C07324=1177.921,389.608,-82.395,-176.029,8.968,148.653
C07325=1177.916,389.855,-82.431,-176.029,8.971,148.654
C07326=1177.913,390.103,-82.467,-176.029,8.974,148.654
C07327=1177.909,390.350,-82.502,-176.028,8.977,148.655
C07328=1177.905,390.597,-82.538,-176.028,8.979,148.656
C07329=1177.901,390.845,-82.573,-176.028,8.983,148.657
C07330=1177.897,391.093,-82.609,-176.027,8.985,148.657
C07331=1177.893,391.340,-82.645,-176.027,8.988,148.658
C07332=1177.889,391.623,-82.686,-176.027,8.991,148.659
C07333=1177.884,391.908,-82.727,-176.027,8.994,148.659
C07334=1177.880,392.193,-82.768,-176.026,8.998,148.660
C07335=1177.874,392.477,-82.808,-176.026,9.001,148.661
C07336=1177.871,392.724,-82.844,-176.026,9.004,148.662
C07337=1177.867,392.972,-82.880,-176.026,9.006,148.662
C07338=1177.863,393.219,-82.915,-176.026,9.009,148.663
C07339=1177.860,393.467,-82.951,-176.026,9.012,148.664
C07340=1177.855,393.714,-82.986,-176.025,9.014,148.664
C07341=1177.851,393.961,-83.023,-176.025,9.017,148.665
C07342=1177.848,394.208,-83.058,-176.025,9.020,148.666
C07343=1177.844,394.456,-83.094,-176.025,9.022,148.666
C07344=1177.840,394.704,-83.130,-176.025,9.025,148.667
C07345=1177.836,394.951,-83.166,-176.025,9.027,148.668
C07346=1177.832,395.198,-83.201,-176.025,9.031,148.668
C07347=1177.827,395.446,-83.237,-176.025,9.033,148.669
C07348=1177.824,395.693,-83.272,-176.025,9.036,148.670
C07349=1177.820,395.941,-83.308,-176.025,9.038,148.670
C07350=1177.816,396.188,-83.343,-176.025,9.040,148.671
C07351=1177.811,396.435,-83.379,-176.025,9.043,148.672
C07352=1177.808,396.682,-83.416,-176.025,9.046,148.672
C07353=1177.804,396.930,-83.451,-176.024,9.049,148.673
C07354=1177.800,397.178,-83.487,-176.024,9.051,148.674
C07355=1177.796,397.425,-83.523,-176.025,9.054,148.674
C07356=1177.793,397.673,-83.558,-176.024,9.056,148.675
C07357=1177.789,397.920,-83.594,-176.024,9.059,148.676
C07358=1177.784,398.167,-83.630,-176.025,9.061,148.676
C07359=1177.780,398.415,-83.665,-176.024,9.064,148.677
C07360=1177.777,398.662,-83.701,-176.024,9.066,148.677
C07361=1177.773,398.909,-83.738,-176.025,9.069,148.678
C07362=1177.769,399.157,-83.773,-176.024,9.071,148.679
C07363=1177.765,399.404,-83.809,-176.025,9.073,148.679
C07364=1177.760,399.652,-83.844,-176.025,9.076,148.680
C07365=1177.757,399.899,-83.880,-176.025,9.077,148.681
C07366=1177.753,400.146,-83.916,-176.025,9.080,148.681
C07367=1177.749,400.394,-83.952,-176.025,9.083,148.682
C07368=1177.745,400.641,-83.988,-176.025,9.085,148.683
C07369=1177.741,400.889,-84.023,-176.025,9.087,148.683
C07370=1177.737,401.137,-84.060,-176.025,9.090,148.684
C07371=1177.733,401.383,-84.096,-176.025,9.092,148.685
C07372=1177.729,401.630,-84.131,-176.025,9.095,148.685
C07373=1177.725,401.878,-84.167,-176.026,9.096,148.686
C07374=1177.721,402.126,-84.203,-176.026,9.099,148.686
C07375=1177.718,402.373,-84.238,-176.026,9.101,148.687
C07376=1177.714,402.620,-84.275,-176.026,9.104,148.688
C07377=1177.710,402.868,-84.311,-176.026,9.106,148.688
C07378=1177.706,403.115,-84.346,-176.026,9.108,148.689
C07379=1177.701,403.362,-84.382,-176.026,9.110,148.690
C07380=1177.698,403.610,-84.418,-176.026,9.113,148.690
C07381=1177.694,403.857,-84.454,-176.026,9.115,148.691
C07382=1177.690,404.105,-84.490,-176.027,9.117,148.691
C07383=1177.686,404.352,-84.526,-176.027,9.119,148.692
C07384=1177.682,404.600,-84.562,-176.027,9.122,148.693
C07385=1177.678,404.847,-84.598,-176.027,9.124,148.693
C07386=1177.675,405.094,-84.634,-176.027,9.126,148.694
C07387=1177.670,405.341,-84.669,-176.027,9.128,148.694
C07388=1177.666,405.589,-84.705,-176.027,9.131,148.695
C07389=1177.663,405.836,-84.741,-176.027,9.132,148.696
C07390=1177.658,406.084,-84.777,-176.028,9.135,148.696
C07391=1177.655,406.331,-84.813,-176.027,9.137,148.697
C07392=1177.651,406.578,-84.850,-176.028,9.139,148.697
C07393=1177.647,406.826,-84.885,-176.028,9.141,148.698
C07394=1177.643,407.073,-84.921,-176.028,9.143,148.699
C07395=1177.639,407.321,-84.957,-176.028,9.145,148.699
C07396=1177.636,407.568,-84.993,-176.028,9.147,148.700
C07397=1177.631,407.815,-85.028,-176.029,9.149,148.700
C07398=1177.627,408.063,-85.064,-176.029,9.151,148.701
C07399=1177.624,408.309,-85.101,-176.029,9.154,148.702
C07400=1177.619,408.557,-85.137,-176.029,9.155,148.702
C07401=1177.615,408.805,-85.172,-176.029,9.158,148.703
C07402=1177.612,409.052,-85.209,-176.030,9.159,148.703
C07403=1177.608,409.299,-85.245,-176.029,9.162,148.704
C07404=1177.604,409.547,-85.280,-176.030,9.163,148.704
C07405=1177.600,409.795,-85.317,-176.030,9.166,148.705
C07406=1177.596,410.042,-85.353,-176.030,9.167,148.706
C07407=1177.592,410.289,-85.389,-176.030,9.170,148.706
C07408=1177.588,410.536,-85.424,-176.030,9.172,148.707
C07409=1177.584,410.783,-85.460,-176.030,9.173,148.707
C07410=1177.580,411.031,-85.497,-176.031,9.176,148.708
C07411=1177.576,411.278,-85.532,-176.031,9.177,148.708
C07412=1177.572,411.526,-85.569,-176.031,9.180,148.709
C07413=1177.568,411.773,-85.604,-176.031,9.181,148.710
C07414=1177.565,412.021,-85.640,-176.031,9.184,148.710
C07415=1177.561,412.268,-85.677,-176.031,9.185,148.711
C07416=1177.557,412.515,-85.712,-176.031,9.188,148.711
C07417=1177.553,412.762,-85.749,-176.032,9.189,148.712
C07418=1177.549,413.010,-85.785,-176.032,9.191,148.712
C07419=1177.545,413.258,-85.821,-176.032,9.193,148.713
C07420=1177.541,413.504,-85.857,-176.033,9.194,148.713
C07421=1177.537,413.752,-85.893,-176.032,9.197,148.714
C07422=1177.533,413.999,-85.929,-176.033,9.198,148.714
C07423=1177.529,414.246,-85.965,-176.033,9.201,148.715
C07424=1177.525,414.494,-86.001,-176.033,9.202,148.715
C07425=1177.522,414.741,-86.037,-176.033,9.204,148.716
C07426=1177.517,414.989,-86.073,-176.033,9.206,148.716
C07427=1177.514,415.236,-86.109,-176.033,9.208,148.717
C07428=1177.510,415.475,-86.144,-176.033,9.210,148.718
C07429=1177.506,415.715,-86.178,-176.034,9.211,148.718
C07430=1177.503,415.955,-86.214,-176.033,9.214,148.719
C07431=1177.502,416.194,-86.248,-176.034,9.215,148.719
C07432=1177.502,416.433,-86.283,-176.034,9.216,148.720
C07433=1177.502,416.672,-86.318,-176.034,9.219,148.720
C07434=1177.505,416.911,-86.352,-176.034,9.220,148.720
C07435=1177.507,417.150,-86.386,-176.034,9.222,148.721
C07436=1177.086,417.151,-86.429,-176.037,9.232,148.725
C07437=1177.083,416.911,-86.395,-176.037,9.231,148.724
C07438=1177.081,416.670,-86.360,-176.037,9.229,148.724
C07439=1177.081,416.430,-86.326,-176.037,9.227,148.723
C07440=1177.081,416.189,-86.291,-176.037,9.226,148.723
C07441=1177.082,415.948,-86.256,-176.036,9.224,148.722
C07442=1177.085,415.707,-86.221,-176.037,9.222,148.722
C07443=1177.088,415.466,-86.186,-176.036,9.221,148.721
C07444=1177.092,415.225,-86.151,-176.036,9.219,148.721
C07445=1177.097,414.977,-86.115,-176.036,9.217,148.720
C07446=1177.100,414.730,-86.079,-176.036,9.215,148.720
C07447=1177.104,414.483,-86.042,-176.036,9.213,148.719
C07448=1177.108,414.235,-86.007,-176.036,9.211,148.719
C07449=1177.112,413.988,-85.970,-176.036,9.209,148.718
C07450=1177.116,413.741,-85.934,-176.036,9.208,148.718
C07451=1177.119,413.493,-85.899,-176.035,9.206,148.717
C07452=1177.123,413.246,-85.862,-176.035,9.204,148.716
C07453=1177.127,412.998,-85.826,-176.035,9.202,148.716
C07454=1177.132,412.751,-85.790,-176.035,9.200,148.715
C07455=1177.135,412.504,-85.754,-176.034,9.198,148.715
C07456=1177.140,412.257,-85.718,-176.035,9.196,148.714
C07457=1177.143,412.010,-85.682,-176.034,9.194,148.714
C07458=1177.148,411.762,-85.646,-176.034,9.192,148.713
C07459=1177.151,411.514,-85.610,-176.034,9.191,148.713
C07460=1177.155,411.267,-85.574,-176.034,9.188,148.712
C07461=1177.159,411.020,-85.538,-176.034,9.187,148.712
C07462=1177.163,410.772,-85.502,-176.034,9.184,148.711
C07463=1177.167,410.525,-85.465,-176.033,9.183,148.710
C07464=1177.170,410.277,-85.430,-176.033,9.180,148.710
C07465=1177.175,410.030,-85.394,-176.033,9.179,148.709
C07466=1177.178,409.783,-85.357,-176.033,9.176,148.709
C07467=1177.182,409.536,-85.322,-176.033,9.175,148.708
C07468=1177.187,409.288,-85.286,-176.032,9.172,148.708
C07469=1177.190,409.041,-85.250,-176.032,9.171,148.707
C07470=1177.195,408.793,-85.214,-176.032,9.168,148.706
C07471=1177.198,408.546,-85.178,-176.032,9.166,148.706
C07472=1177.202,408.299,-85.142,-176.032,9.164,148.705
C07473=1177.206,408.051,-85.106,-176.032,9.162,148.705
C07474=1177.210,407.804,-85.070,-176.031,9.160,148.704
C07475=1177.214,407.557,-85.033,-176.031,9.158,148.703
C07476=1177.217,407.309,-84.998,-176.032,9.156,148.703
C07477=1177.221,407.062,-84.962,-176.031,9.154,148.702
C07478=1177.226,406.815,-84.926,-176.031,9.152,148.702
C07479=1177.230,406.568,-84.890,-176.030,9.150,148.701
C07480=1177.234,406.320,-84.854,-176.031,9.148,148.701
C07481=1177.238,406.072,-84.818,-176.031,9.145,148.700
C07482=1177.241,405.825,-84.782,-176.030,9.143,148.699
C07483=1177.245,405.578,-84.746,-176.030,9.141,148.699
C07484=1177.249,405.330,-84.710,-176.030,9.139,148.698
C07485=1177.253,405.082,-84.674,-176.030,9.137,148.698
C07486=1177.257,404.835,-84.638,-176.029,9.135,148.697
C07487=1177.261,404.589,-84.603,-176.030,9.132,148.696
C07488=1177.265,404.341,-84.567,-176.029,9.131,148.696
C07489=1177.269,404.093,-84.531,-176.029,9.128,148.695
C07490=1177.272,403.846,-84.495,-176.029,9.126,148.694
C07491=1177.277,403.599,-84.459,-176.029,9.123,148.694
C07492=1177.281,403.351,-84.423,-176.029,9.122,148.693
C07493=1177.285,403.103,-84.387,-176.029,9.119,148.693
C07494=1177.288,402.856,-84.351,-176.029,9.117,148.692
C07495=1177.292,402.609,-84.315,-176.029,9.114,148.691
C07496=1177.297,402.362,-84.279,-176.028,9.113,148.691
C07497=1177.301,402.114,-84.244,-176.028,9.110,148.690
C07498=1177.304,401.867,-84.208,-176.028,9.108,148.689
C07499=1177.308,401.620,-84.172,-176.028,9.106,148.689
C07500=1177.312,401.372,-84.136,-176.028,9.103,148.688
C07501=1177.316,401.125,-84.100,-176.027,9.101,148.687
C07502=1177.320,400.877,-84.064,-176.028,9.099,148.687
C07503=1177.324,400.631,-84.028,-176.027,9.096,148.686
C07504=1177.328,400.383,-83.993,-176.027,9.094,148.686
C07505=1177.332,400.135,-83.957,-176.028,9.092,148.685
C07506=1177.336,399.888,-83.921,-176.027,9.089,148.684
C07507=1177.339,399.640,-83.886,-176.027,9.086,148.684
C07508=1177.344,399.393,-83.849,-176.028,9.084,148.683
C07509=1177.347,399.146,-83.813,-176.027,9.082,148.682
C07510=1177.351,398.898,-83.778,-176.027,9.079,148.682
C07511=1177.356,398.651,-83.742,-176.027,9.077,148.681
C07512=1177.359,398.404,-83.706,-176.027,9.074,148.680
C07513=1177.363,398.156,-83.671,-176.027,9.072,148.680
C07514=1177.367,397.909,-83.634,-176.027,9.069,148.679
C07515=1177.371,397.661,-83.598,-176.027,9.067,148.678
C07516=1177.375,397.414,-83.563,-176.027,9.064,148.678
C07517=1177.380,397.167,-83.527,-176.027,9.062,148.677
C07518=1177.383,396.919,-83.491,-176.027,9.059,148.676
C07519=1177.387,396.672,-83.456,-176.027,9.057,148.676
C07520=1177.391,396.424,-83.420,-176.027,9.054,148.675
C07521=1177.395,396.177,-83.384,-176.027,9.052,148.675
C07522=1177.398,395.930,-83.348,-176.027,9.049,148.674
C07523=1177.403,395.683,-83.313,-176.027,9.047,148.673
C07524=1177.407,395.435,-83.277,-176.027,9.045,148.673
C07525=1177.411,395.187,-83.241,-176.027,9.041,148.672
C07526=1177.414,394.940,-83.206,-176.027,9.039,148.671
C07527=1177.418,394.692,-83.170,-176.027,9.036,148.670
C07528=1177.422,394.445,-83.134,-176.027,9.034,148.670
C07529=1177.427,394.198,-83.099,-176.027,9.031,148.669
C07530=1177.430,393.950,-83.063,-176.028,9.028,148.668
C07531=1177.434,393.703,-83.027,-176.028,9.026,148.668
C07532=1177.438,393.456,-82.991,-176.028,9.023,148.667
C07533=1177.442,393.208,-82.955,-176.028,9.020,148.666
C07534=1177.445,392.961,-82.920,-176.028,9.017,148.666
C07535=1177.450,392.714,-82.884,-176.028,9.015,148.665
C07536=1177.454,392.466,-82.848,-176.028,9.012,148.664
C07537=1177.458,392.181,-82.808,-176.028,9.009,148.664
C07538=1177.463,391.897,-82.766,-176.029,9.005,148.663
C07539=1177.467,391.613,-82.726,-176.029,9.002,148.662
C07540=1177.472,391.328,-82.684,-176.029,8.999,148.661
C07541=1177.476,391.081,-82.649,-176.029,8.996,148.661
C07542=1177.479,390.833,-82.613,-176.030,8.994,148.660
C07543=1177.484,390.587,-82.578,-176.030,8.990,148.659
C07544=1177.487,390.339,-82.543,-176.030,8.988,148.659
C07545=1177.492,390.091,-82.506,-176.031,8.985,148.658
C07546=1177.495,389.844,-82.471,-176.031,8.982,148.657
C07547=1177.499,389.596,-82.435,-176.031,8.979,148.657
C07548=1177.503,389.350,-82.400,-176.031,8.977,148.656
C07549=1177.507,389.102,-82.365,-176.032,8.973,148.655
C07550=1177.511,388.854,-82.328,-176.033,8.970,148.655
C07551=1177.515,388.607,-82.293,-176.032,8.967,148.654
C07552=1177.519,388.360,-82.258,-176.033,8.964,148.653
C07553=1177.523,388.112,-82.223,-176.034,8.961,148.652
C07554=1177.527,387.864,-82.187,-176.034,8.959,148.652
C07555=1177.531,387.617,-82.152,-176.034,8.955,148.651
C07556=1177.535,387.369,-82.116,-176.035,8.952,148.651
C07557=1177.539,387.122,-82.080,-176.035,8.949,148.650
C07558=1177.543,386.875,-82.045,-176.036,8.947,148.649
C07559=1177.547,386.627,-82.009,-176.036,8.943,148.649
C07560=1177.550,386.380,-81.974,-176.037,8.940,148.648
C07561=1177.554,386.133,-81.939,-176.037,8.937,148.647
C07562=1177.558,385.885,-81.903,-176.038,8.934,148.647
C07563=1177.563,385.637,-81.868,-176.038,8.931,148.646
C07564=1177.567,385.390,-81.832,-176.039,8.928,148.645
C07565=1177.571,385.143,-81.797,-176.040,8.925,148.645
C07566=1177.574,384.895,-81.761,-176.040,8.921,148.644
C07567=1177.578,384.648,-81.726,-176.041,8.918,148.643
C07568=1177.582,384.401,-81.691,-176.042,8.915,148.643
C07569=1177.586,384.153,-81.655,-176.042,8.912,148.642
C07570=1177.590,383.905,-81.620,-176.043,8.909,148.641
C07571=1177.594,383.658,-81.585,-176.044,8.906,148.641
C07572=1177.599,383.411,-81.549,-176.044,8.902,148.640
C07573=1177.602,383.163,-81.513,-176.045,8.899,148.639
C07574=1177.606,382.915,-81.479,-176.046,8.896,148.639
C07575=1177.610,382.668,-81.443,-176.047,8.892,148.638
C07576=1177.614,382.421,-81.408,-176.048,8.889,148.637
C07577=1177.618,382.173,-81.372,-176.048,8.886,148.637
C07578=1177.622,381.926,-81.337,-176.049,8.883,148.636
C07579=1177.626,381.678,-81.302,-176.050,8.880,148.636
C07580=1177.630,381.431,-81.267,-176.051,8.876,148.635
C07581=1177.633,381.183,-81.231,-176.052,8.873,148.635
C07582=1177.638,380.936,-81.197,-176.053,8.869,148.634
C07583=1177.642,380.688,-81.161,-176.054,8.866,148.633
C07584=1177.645,380.441,-81.126,-176.054,8.863,148.633
C07585=1177.650,380.194,-81.091,-176.056,8.859,148.632
C07586=1177.654,379.946,-81.056,-176.057,8.856,148.631
C07587=1177.657,379.698,-81.020,-176.057,8.853,148.631
C07588=1177.662,379.451,-80.986,-176.059,8.849,148.630
C07589=1177.665,379.204,-80.950,-176.060,8.846,148.630
C07590=1177.669,378.956,-80.914,-176.060,8.843,148.629
C07591=1177.674,378.709,-80.880,-176.062,8.839,148.628
C07592=1177.677,378.461,-80.844,-176.063,8.836,148.628
C07593=1177.681,378.214,-80.809,-176.064,8.832,148.627
C07594=1177.686,377.966,-80.774,-176.065,8.829,148.627
C07595=1177.689,377.719,-80.739,-176.066,8.825,148.626
C07596=1177.693,377.471,-80.704,-176.068,8.822,148.626
C07597=1177.697,377.224,-80.669,-176.068,8.819,148.625
C07598=1177.701,376.976,-80.634,-176.070,8.815,148.624
C07599=1177.705,376.728,-80.598,-176.071,8.812,148.624
C07600=1177.709,376.481,-80.563,-176.072,8.808,148.623
C07601=1177.713,376.233,-80.528,-176.074,8.804,148.623
C07602=1177.718,375.986,-80.493,-176.075,8.801,148.622
C07603=1177.722,375.738,-80.458,-176.076,8.797,148.622
C07604=1177.724,375.491,-80.423,-176.077,8.794,148.621
C07605=1177.729,375.244,-80.389,-176.079,8.791,148.621
C07606=1177.733,374.996,-80.353,-176.080,8.788,148.620
C07607=1177.737,374.749,-80.319,-176.081,8.784,148.619
C07608=1177.741,374.501,-80.283,-176.083,8.780,148.619
C07609=1177.745,374.253,-80.249,-176.084,8.777,148.618
C07610=1177.749,374.006,-80.214,-176.085,8.773,148.618
C07611=1177.753,373.758,-80.179,-176.087,8.769,148.617
C07612=1177.757,373.511,-80.145,-176.088,8.766,148.617
C07613=1177.761,373.264,-80.109,-176.089,8.763,148.616
C07614=1177.765,373.016,-80.074,-176.091,8.759,148.616
C07615=1177.769,372.768,-80.040,-176.092,8.756,148.615
C07616=1177.773,372.521,-80.004,-176.094,8.752,148.615
C07617=1177.777,372.273,-79.970,-176.095,8.748,148.614
C07618=1177.780,372.026,-79.935,-176.097,8.745,148.613
C07619=1177.785,371.779,-79.900,-176.099,8.741,148.613
C07620=1177.789,371.530,-79.866,-176.099,8.738,148.612
C07621=1177.793,371.282,-79.831,-176.101,8.734,148.612
C07622=1177.797,371.036,-79.796,-176.103,8.731,148.612
C07623=1177.800,370.788,-79.761,-176.104,8.727,148.611
C07624=1177.805,370.540,-79.727,-176.106,8.723,148.611
C07625=1177.809,370.293,-79.691,-176.108,8.720,148.610
C07626=1177.813,370.045,-79.657,-176.109,8.716,148.610
C07627=1177.816,369.798,-79.623,-176.111,8.713,148.609
C07628=1177.821,369.550,-79.588,-176.113,8.709,148.609
C07629=1177.825,369.303,-79.553,-176.114,8.706,148.608
C07630=1177.829,369.055,-79.518,-176.116,8.702,148.608
C07631=1177.832,368.807,-79.484,-176.118,8.698,148.607
C07632=1177.837,368.560,-79.449,-176.119,8.695,148.607
C07633=1177.841,368.312,-79.415,-176.121,8.692,148.606
C07634=1177.844,368.065,-79.380,-176.123,8.688,148.606
C07635=1177.848,367.817,-79.345,-176.124,8.684,148.606
C07636=1177.853,367.570,-79.311,-176.126,8.681,148.605
C07637=1177.856,367.322,-79.277,-176.128,8.677,148.605
C07638=1177.861,367.075,-79.242,-176.130,8.674,148.604
C07639=1177.865,366.827,-79.207,-176.132,8.670,148.604
C07640=1177.869,366.579,-79.173,-176.134,8.666,148.603
C07641=1177.873,366.298,-79.134,-176.135,8.662,148.603
C07642=1177.878,366.016,-79.094,-176.137,8.658,148.602
C07643=1177.882,365.734,-79.055,-176.140,8.653,148.602
C07644=1177.887,365.452,-79.016,-176.142,8.650,148.601
C07645=1177.891,365.205,-78.981,-176.143,8.646,148.601
C07646=1177.895,364.957,-78.947,-176.145,8.643,148.600
C07647=1177.899,364.710,-78.913,-176.147,8.639,148.600
C07648=1177.902,364.462,-78.878,-176.149,8.636,148.600
C07649=1177.907,364.215,-78.844,-176.151,8.632,148.599
C07650=1177.911,363.968,-78.810,-176.153,8.628,148.599
C07651=1177.915,363.719,-78.775,-176.155,8.625,148.599
C07652=1177.919,363.472,-78.741,-176.157,8.622,148.598
C07653=1177.923,363.224,-78.707,-176.159,8.618,148.598
C07654=1177.927,362.976,-78.673,-176.161,8.614,148.597
C07655=1177.931,362.729,-78.639,-176.163,8.611,148.597
C07656=1177.935,362.481,-78.604,-176.165,8.607,148.597
C07657=1177.939,362.234,-78.570,-176.167,8.603,148.596
C07658=1177.943,361.986,-78.535,-176.169,8.599,148.596
C07659=1177.947,361.739,-78.501,-176.171,8.596,148.596
C07660=1177.951,361.491,-78.467,-176.173,8.592,148.595
C07661=1177.955,361.243,-78.433,-176.175,8.589,148.595
C07662=1177.960,360.995,-78.399,-176.177,8.585,148.595
C07663=1177.963,360.748,-78.365,-176.179,8.582,148.594
C07664=1177.967,360.500,-78.331,-176.181,8.579,148.594
C07665=1177.971,360.253,-78.296,-176.183,8.575,148.593
C07666=1177.975,360.005,-78.263,-176.185,8.572,148.593
C07667=1177.979,359.757,-78.228,-176.188,8.567,148.593
C07668=1177.983,359.510,-78.195,-176.190,8.564,148.593
C07669=1177.988,359.263,-78.160,-176.192,8.560,148.592
C07670=1177.991,359.014,-78.127,-176.194,8.557,148.592
C07671=1177.995,358.767,-78.093,-176.196,8.553,148.591
C07672=1178.000,358.520,-78.058,-176.198,8.550,148.591
C07673=1178.003,358.271,-78.025,-176.200,8.546,148.591
C07674=1178.008,358.024,-77.990,-176.202,8.543,148.591
C07675=1178.012,357.777,-77.956,-176.205,8.539,148.590
C07676=1178.015,357.528,-77.923,-176.207,8.535,148.590
C07677=1178.020,357.281,-77.888,-176.209,8.532,148.590
C07678=1178.024,357.033,-77.855,-176.211,8.528,148.589
C07679=1178.028,356.786,-77.821,-176.213,8.525,148.589
C07680=1178.032,356.538,-77.787,-176.216,8.522,148.589
C07681=1178.036,356.290,-77.753,-176.217,8.518,148.588
C07682=1178.040,356.043,-77.720,-176.220,8.514,148.588
C07683=1178.044,355.794,-77.685,-176.223,8.511,148.588
C07684=1178.048,355.547,-77.652,-176.224,8.507,148.587
C07685=1178.052,355.299,-77.618,-176.227,8.504,148.587
C07686=1178.056,355.052,-77.584,-176.229,8.501,148.587
C07687=1178.060,354.804,-77.550,-176.231,8.497,148.587
C07688=1178.064,354.556,-77.517,-176.233,8.494,148.586
C07689=1178.068,354.309,-77.483,-176.235,8.490,148.586
C07690=1178.072,354.062,-77.449,-176.238,8.486,148.586
C07691=1178.077,353.814,-77.416,-176.240,8.483,148.586
C07692=1178.080,353.565,-77.382,-176.242,8.479,148.585
C07693=1178.084,353.318,-77.348,-176.245,8.476,148.585
C07694=1178.088,353.070,-77.315,-176.247,8.473,148.585
C07695=1178.093,352.823,-77.281,-176.249,8.469,148.585
C07696=1178.097,352.575,-77.248,-176.251,8.466,148.584
C07697=1178.100,352.327,-77.214,-176.253,8.462,148.584
C07698=1178.104,352.080,-77.180,-176.256,8.458,148.584
C07699=1178.108,351.832,-77.147,-176.258,8.455,148.583
C07700=1178.113,351.584,-77.113,-176.261,8.452,148.583
C07701=1178.117,351.337,-77.079,-176.262,8.448,148.583
C07702=1178.121,351.089,-77.046,-176.265,8.445,148.583
C07703=1178.125,350.841,-77.013,-176.267,8.441,148.582
C07704=1178.129,350.593,-76.980,-176.269,8.438,148.582
C07705=1178.133,350.346,-76.946,-176.271,8.435,148.582
C07706=1178.137,350.098,-76.913,-176.274,8.431,148.582
C07707=1178.141,349.850,-76.879,-176.277,8.427,148.581
C07708=1178.146,349.602,-76.846,-176.279,8.424,148.581
C07709=1178.150,349.355,-76.812,-176.281,8.420,148.581
C07710=1178.153,349.107,-76.778,-176.283,8.417,148.581
C07711=1178.157,348.859,-76.745,-176.285,8.414,148.580
C07712=1178.161,348.611,-76.712,-176.287,8.410,148.580
C07713=1178.166,348.364,-76.679,-176.290,8.407,148.580
C07714=1178.170,348.116,-76.646,-176.292,8.404,148.580
C07715=1178.174,347.868,-76.612,-176.294,8.401,148.579
C07716=1178.178,347.620,-76.579,-176.296,8.397,148.579
C07717=1178.182,347.373,-76.545,-176.299,8.393,148.579
C07718=1178.186,347.125,-76.512,-176.302,8.390,148.579
C07719=1178.190,346.878,-76.479,-176.304,8.386,148.579
C07720=1178.194,346.630,-76.446,-176.306,8.383,148.578
C07721=1178.198,346.382,-76.413,-176.308,8.380,148.578
C07722=1178.202,346.134,-76.379,-176.311,8.377,148.578
C07723=1178.206,345.886,-76.346,-176.313,8.373,148.578
C07724=1178.210,345.638,-76.313,-176.315,8.370,148.577
C07725=1178.214,345.391,-76.280,-176.317,8.367,148.577
C07726=1178.219,345.143,-76.247,-176.320,8.363,148.577
C07727=1178.223,344.895,-76.214,-176.322,8.360,148.577
C07728=1178.227,344.647,-76.180,-176.324,8.357,148.577
C07729=1178.231,344.399,-76.148,-176.327,8.353,148.576
C07730=1178.235,344.151,-76.115,-176.329,8.349,148.576
C07731=1178.240,343.904,-76.082,-176.332,8.346,148.576
C07732=1178.244,343.656,-76.048,-176.334,8.343,148.576
C07733=1178.248,343.408,-76.015,-176.336,8.339,148.576
C07734=1178.252,343.160,-75.982,-176.338,8.336,148.575
C07735=1178.255,342.913,-75.950,-176.341,8.333,148.575
C07736=1178.259,342.665,-75.916,-176.343,8.329,148.575
C07737=1178.264,342.417,-75.884,-176.345,8.326,148.575
C07738=1178.268,342.169,-75.851,-176.348,8.323,148.575
C07739=1178.272,341.922,-75.818,-176.350,8.320,148.574
C07740=1178.276,341.674,-75.785,-176.353,8.316,148.574
C07741=1178.281,341.425,-75.752,-176.355,8.313,148.574
C07742=1178.284,341.178,-75.719,-176.357,8.310,148.574
C07743=1178.289,340.931,-75.687,-176.359,8.307,148.574
C07744=1178.293,340.683,-75.654,-176.362,8.302,148.573
C07745=1178.298,340.404,-75.616,-176.364,8.299,148.573
C07746=1178.302,340.125,-75.580,-176.368,8.295,148.573
C07747=1178.307,339.845,-75.543,-176.370,8.292,148.573
C07748=1178.311,339.566,-75.506,-176.373,8.288,148.573
C07749=1178.316,339.319,-75.473,-176.375,8.285,148.572
C07750=1178.320,339.070,-75.440,-176.377,8.281,148.572
C07751=1178.323,338.823,-75.408,-176.380,8.278,148.572
C07752=1178.328,338.575,-75.375,-176.382,8.275,148.572
C07753=1178.332,338.327,-75.342,-176.385,8.272,148.572
C07754=1178.336,338.079,-75.309,-176.387,8.268,148.572
C07755=1178.340,337.832,-75.278,-176.389,8.265,148.571
C07756=1178.345,337.584,-75.245,-176.391,8.262,148.571
C07757=1178.349,337.336,-75.212,-176.394,8.259,148.571
C07758=1178.352,337.088,-75.180,-176.396,8.255,148.571
C07759=1178.357,336.841,-75.146,-176.399,8.252,148.571
C07760=1178.361,336.592,-75.114,-176.401,8.249,148.570
C07761=1178.364,336.345,-75.081,-176.404,8.246,148.570
C07762=1178.369,336.096,-75.049,-176.406,8.242,148.570
C07763=1178.374,335.849,-75.016,-176.409,8.238,148.570
C07764=1178.377,335.601,-74.984,-176.411,8.235,148.570
C07765=1178.382,335.353,-74.952,-176.414,8.232,148.570
C07766=1178.385,335.106,-74.919,-176.416,8.229,148.570
C07767=1178.390,334.857,-74.887,-176.418,8.225,148.569
C07768=1178.394,334.609,-74.854,-176.421,8.222,148.569
C07769=1178.398,334.362,-74.822,-176.423,8.219,148.569
C07770=1178.403,334.114,-74.790,-176.426,8.216,148.569
C07771=1178.406,333.866,-74.757,-176.428,8.212,148.569
C07772=1178.410,333.618,-74.725,-176.430,8.209,148.569
C07773=1178.414,333.370,-74.693,-176.433,8.206,148.569
C07774=1178.419,333.123,-74.660,-176.435,8.203,148.568
C07775=1178.423,332.875,-74.628,-176.437,8.200,148.568
C07776=1178.427,332.627,-74.596,-176.440,8.197,148.568
C07777=1178.431,332.379,-74.563,-176.442,8.193,148.568
C07778=1178.435,332.131,-74.531,-176.445,8.190,148.568
C07779=1178.440,331.883,-74.499,-176.447,8.187,148.568
C07780=1178.444,331.635,-74.467,-176.450,8.184,148.567
C07781=1178.448,331.387,-74.434,-176.452,8.180,148.567
C07782=1178.451,331.139,-74.402,-176.455,8.177,148.567
C07783=1178.456,330.892,-74.370,-176.457,8.174,148.567
C07784=1178.460,330.644,-74.338,-176.459,8.171,148.567
C07785=1178.465,330.395,-74.306,-176.462,8.168,148.567
C07786=1178.468,330.148,-74.273,-176.464,8.164,148.567
C07787=1178.472,329.901,-74.242,-176.466,8.161,148.566
C07788=1178.477,329.652,-74.209,-176.469,8.158,148.566
C07789=1178.480,329.404,-74.177,-176.471,8.155,148.566
C07790=1178.485,329.156,-74.145,-176.474,8.152,148.566
C07791=1178.489,328.908,-74.113,-176.476,8.148,148.566
C07792=1178.493,328.660,-74.081,-176.479,8.145,148.566
C07793=1178.497,328.412,-74.049,-176.481,8.142,148.566
C07794=1178.502,328.165,-74.018,-176.484,8.139,148.566
C07795=1178.506,327.916,-73.985,-176.486,8.136,148.566
C07796=1178.510,327.668,-73.953,-176.489,8.133,148.565
C07797=1178.514,327.421,-73.922,-176.491,8.129,148.565
C07798=1178.519,327.173,-73.889,-176.494,8.126,148.565
C07799=1178.522,326.925,-73.858,-176.496,8.123,148.565
C07800=1178.527,326.677,-73.826,-176.498,8.120,148.565
C07801=1178.531,326.429,-73.794,-176.501,8.117,148.565
C07802=1178.535,326.181,-73.762,-176.503,8.114,148.565
C07803=1178.539,325.934,-73.730,-176.506,8.110,148.565
C07804=1178.543,325.685,-73.698,-176.508,8.107,148.564
C07805=1178.547,325.437,-73.666,-176.511,8.104,148.564
C07806=1178.551,325.190,-73.635,-176.513,8.101,148.564
C07807=1178.555,324.942,-73.603,-176.516,8.098,148.564
C07808=1178.560,324.693,-73.570,-176.518,8.094,148.564
C07809=1178.564,324.446,-73.539,-176.521,8.091,148.564
C07810=1178.568,324.197,-73.508,-176.523,8.088,148.564
C07811=1178.572,323.949,-73.476,-176.526,8.085,148.564
C07812=1178.577,323.702,-73.444,-176.528,8.082,148.564
C07813=1178.580,323.454,-73.412,-176.531,8.079,148.564
C07814=1178.585,323.206,-73.380,-176.533,8.075,148.563
C07815=1178.588,322.958,-73.349,-176.536,8.072,148.563
C07816=1178.592,322.710,-73.317,-176.538,8.069,148.563
C07817=1178.597,322.462,-73.285,-176.541,8.066,148.563
C07818=1178.601,322.214,-73.253,-176.543,8.063,148.563
C07819=1178.605,321.967,-73.222,-176.546,8.060,148.563
C07820=1178.610,321.718,-73.191,-176.548,8.057,148.563
C07821=1178.614,321.471,-73.159,-176.551,8.054,148.563
C07822=1178.618,321.223,-73.128,-176.553,8.050,148.563
C07823=1178.622,320.974,-73.096,-176.556,8.047,148.563
C07824=1178.627,320.726,-73.064,-176.558,8.044,148.562
C07825=1178.630,320.478,-73.032,-176.561,8.041,148.562
C07826=1178.635,320.230,-73.002,-176.563,8.038,148.562
C07827=1178.639,319.982,-72.970,-176.566,8.035,148.562
C07828=1178.643,319.734,-72.939,-176.568,8.031,148.562
C07829=1178.647,319.486,-72.907,-176.571,8.028,148.562
C07830=1178.651,319.239,-72.876,-176.573,8.025,148.562
C07831=1178.655,318.990,-72.845,-176.576,8.022,148.562
C07832=1178.660,318.743,-72.813,-176.578,8.019,148.562
C07833=1178.664,318.494,-72.782,-176.581,8.016,148.562
C07834=1178.668,318.247,-72.751,-176.583,8.012,148.561
C07835=1178.672,317.998,-72.719,-176.586,8.009,148.562
C07836=1178.676,317.751,-72.688,-176.588,8.007,148.562
C07837=1178.680,317.502,-72.657,-176.590,8.004,148.561
C07838=1178.685,317.255,-72.625,-176.593,8.001,148.561
C07839=1178.689,317.006,-72.594,-176.595,7.998,148.561
C07840=1178.693,316.759,-72.563,-176.598,7.995,148.561
C07841=1178.697,316.510,-72.532,-176.600,7.991,148.561
C07842=1178.701,316.263,-72.500,-176.603,7.988,148.561
C07843=1178.705,316.014,-72.469,-176.605,7.985,148.561
C07844=1178.710,315.766,-72.438,-176.608,7.982,148.561
C07845=1178.714,315.519,-72.407,-176.610,7.979,148.561
C07846=1178.718,315.270,-72.376,-176.613,7.976,148.561
C07847=1178.723,315.022,-72.345,-176.615,7.973,148.561
C07848=1178.726,314.774,-72.313,-176.618,7.970,148.561
C07849=1178.731,314.498,-72.278,-176.620,7.966,148.560
C07850=1178.736,314.220,-72.244,-176.624,7.963,148.560
C07851=1178.741,313.945,-72.210,-176.626,7.960,148.560
C07852=1178.746,313.668,-72.174,-176.629,7.956,148.560
C07853=1178.750,313.419,-72.143,-176.631,7.953,148.560
C07854=1178.754,313.171,-72.112,-176.634,7.950,148.560
C07855=1178.758,312.924,-72.082,-176.636,7.947,148.560
C07856=1178.762,312.676,-72.050,-176.639,7.944,148.560
C07857=1178.766,312.428,-72.020,-176.642,7.941,148.560
C07858=1178.770,312.179,-71.989,-176.644,7.938,148.560
C07859=1178.775,311.931,-71.958,-176.647,7.935,148.560
C07860=1178.780,311.683,-71.927,-176.649,7.931,148.560
C07861=1178.783,311.435,-71.895,-176.652,7.928,148.560
C07862=1178.787,311.187,-71.865,-176.655,7.925,148.560
C07863=1178.792,310.939,-71.834,-176.657,7.922,148.560
C07864=1178.796,310.691,-71.803,-176.659,7.919,148.560
C07865=1178.800,310.443,-71.772,-176.662,7.916,148.560
C07866=1178.804,310.195,-71.742,-176.664,7.913,148.559
C07867=1178.808,309.946,-71.711,-176.667,7.910,148.559
C07868=1178.813,309.698,-71.680,-176.669,7.908,148.559
C07869=1178.818,309.451,-71.650,-176.672,7.904,148.559
C07870=1178.821,309.202,-71.619,-176.674,7.901,148.559
C07871=1178.825,308.954,-71.588,-176.677,7.898,148.559
C07872=1178.830,308.706,-71.557,-176.679,7.895,148.559
C07873=1178.835,308.458,-71.527,-176.682,7.892,148.559
C07874=1178.838,308.210,-71.496,-176.685,7.889,148.559
C07875=1178.843,307.962,-71.465,-176.688,7.886,148.559
C07876=1178.847,307.714,-71.435,-176.690,7.883,148.559
C07877=1178.850,307.466,-71.404,-176.693,7.880,148.559
C07878=1178.855,307.218,-71.373,-176.695,7.877,148.559
C07879=1178.860,306.970,-71.343,-176.697,7.874,148.559
C07880=1178.863,306.722,-71.312,-176.700,7.871,148.559
C07881=1178.868,306.473,-71.281,-176.702,7.868,148.559
C07882=1178.872,306.225,-71.250,-176.705,7.865,148.559
C07883=1178.876,305.978,-71.220,-176.707,7.862,148.559
C07884=1178.881,305.730,-71.190,-176.710,7.859,148.559
C07885=1178.885,305.481,-71.159,-176.713,7.856,148.559
C07886=1178.889,305.233,-71.129,-176.715,7.853,148.559
C07887=1178.893,304.985,-71.098,-176.718,7.850,148.559
C07888=1178.897,304.737,-71.068,-176.721,7.847,148.559
C07889=1178.902,304.489,-71.037,-176.723,7.844,148.558
C07890=1178.906,304.240,-71.007,-176.726,7.841,148.558
C07891=1178.910,303.992,-70.977,-176.728,7.838,148.559
C07892=1178.915,303.745,-70.946,-176.730,7.835,148.559
C07893=1178.919,303.497,-70.916,-176.733,7.832,148.558
C07894=1178.924,303.248,-70.886,-176.735,7.829,148.558
C07895=1178.927,303.000,-70.855,-176.738,7.826,148.558
C07896=1178.931,302.752,-70.824,-176.741,7.823,148.558
C07897=1178.935,302.504,-70.794,-176.743,7.820,148.558
C07898=1178.940,302.256,-70.764,-176.746,7.817,148.558
C07899=1178.945,302.008,-70.733,-176.749,7.814,148.558
C07900=1178.949,301.760,-70.704,-176.751,7.812,148.558
C07901=1178.953,301.512,-70.674,-176.753,7.808,148.558
C07902=1178.957,301.263,-70.643,-176.756,7.805,148.558
C07903=1178.961,301.015,-70.613,-176.758,7.802,148.558
C07904=1178.966,300.767,-70.582,-176.761,7.799,148.558
C07905=1178.970,300.519,-70.552,-176.764,7.796,148.558
C07906=1178.974,300.271,-70.522,-176.766,7.793,148.558
C07907=1178.978,300.023,-70.492,-176.769,7.790,148.558
C07908=1178.983,299.775,-70.462,-176.772,7.787,148.558
C07909=1178.987,299.526,-70.431,-176.774,7.785,148.558
C07910=1178.991,299.278,-70.402,-176.776,7.782,148.558
C07911=1178.995,299.030,-70.371,-176.779,7.779,148.558
C07912=1179.000,298.782,-70.342,-176.782,7.776,148.558
C07913=1179.004,298.534,-70.311,-176.784,7.773,148.558
C07914=1179.008,298.285,-70.282,-176.787,7.770,148.558
C07915=1179.012,298.038,-70.251,-176.789,7.766,148.558
C07916=1179.017,297.789,-70.221,-176.792,7.763,148.558
C07917=1179.021,297.541,-70.192,-176.794,7.761,148.558
C07918=1179.025,297.293,-70.162,-176.797,7.758,148.558
C07919=1179.030,297.045,-70.132,-176.800,7.755,148.558
C07920=1179.034,296.797,-70.102,-176.802,7.752,148.558
C07921=1179.038,296.549,-70.072,-176.805,7.749,148.558
C07922=1179.042,296.300,-70.042,-176.807,7.746,148.558
C07923=1179.046,296.052,-70.012,-176.810,7.743,148.558
C07924=1179.051,295.804,-69.982,-176.812,7.741,148.558
C07925=1179.055,295.555,-69.953,-176.815,7.738,148.558
C07926=1179.059,295.307,-69.922,-176.817,7.735,148.558
C07927=1179.063,295.059,-69.892,-176.820,7.732,148.558
C07928=1179.068,294.811,-69.863,-176.823,7.729,148.558
C07929=1179.072,294.563,-69.833,-176.825,7.726,148.558
C07930=1179.076,294.315,-69.803,-176.828,7.723,148.558
C07931=1179.081,294.066,-69.773,-176.830,7.720,148.558
C07932=1179.085,293.818,-69.744,-176.833,7.717,148.558
C07933=1179.089,293.570,-69.714,-176.835,7.714,148.558
C07934=1179.093,293.322,-69.684,-176.838,7.711,148.558
C07935=1179.098,293.074,-69.654,-176.841,7.708,148.558
C07936=1179.102,292.825,-69.625,-176.843,7.705,148.558
C07937=1179.106,292.577,-69.595,-176.846,7.703,148.558
C07938=1179.110,292.329,-69.566,-176.848,7.700,148.558
C07939=1179.114,292.081,-69.536,-176.851,7.697,148.558
C07940=1179.118,291.833,-69.506,-176.853,7.694,148.558
C07941=1179.123,291.584,-69.476,-176.856,7.691,148.558
C07942=1179.128,291.337,-69.447,-176.859,7.688,148.558
C07943=1179.132,291.089,-69.418,-176.861,7.686,148.558
C07944=1179.136,290.840,-69.388,-176.864,7.683,148.558
C07945=1179.141,290.592,-69.359,-176.866,7.680,148.558
C07946=1179.145,290.344,-69.329,-176.869,7.677,148.558
C07947=1179.149,290.095,-69.300,-176.871,7.673,148.558
C07948=1179.153,289.847,-69.270,-176.874,7.670,148.558
C07949=1179.157,289.599,-69.241,-176.876,7.668,148.558
C07950=1179.162,289.351,-69.211,-176.879,7.665,148.558
C07951=1179.166,289.102,-69.182,-176.882,7.662,148.558
C07952=1179.171,288.854,-69.152,-176.884,7.659,148.558
C07953=1179.175,288.580,-69.120,-176.887,7.656,148.558
C07954=1179.180,288.305,-69.087,-176.890,7.653,148.558
C07955=1179.185,288.031,-69.055,-176.893,7.649,148.558
C07956=1179.190,287.756,-69.022,-176.896,7.646,148.558
C07957=1179.194,287.507,-68.993,-176.899,7.643,148.558
C07958=1179.198,287.259,-68.963,-176.901,7.641,148.558
C07959=1179.202,287.011,-68.934,-176.904,7.638,148.558
C07960=1179.207,286.763,-68.905,-176.906,7.635,148.558
C07961=1179.211,286.514,-68.876,-176.909,7.632,148.558
C07962=1179.216,286.266,-68.846,-176.911,7.629,148.558
C07963=1179.220,286.018,-68.817,-176.913,7.627,148.558
C07964=1179.224,285.769,-68.787,-176.916,7.624,148.558
C07965=1179.228,285.521,-68.758,-176.919,7.621,148.558
C07966=1179.233,285.273,-68.730,-176.922,7.618,148.558
C07967=1179.237,285.025,-68.700,-176.924,7.615,148.558
C07968=1179.241,284.777,-68.671,-176.927,7.613,148.559
C07969=1179.245,284.529,-68.642,-176.929,7.610,148.559
C07970=1179.249,284.280,-68.613,-176.932,7.607,148.559
C07971=1179.254,284.032,-68.584,-176.935,7.604,148.559
C07972=1179.258,283.784,-68.555,-176.937,7.601,148.559
C07973=1179.263,283.535,-68.526,-176.940,7.599,148.559
C07974=1179.267,283.287,-68.496,-176.942,7.596,148.559
C07975=1179.271,283.038,-68.467,-176.945,7.593,148.559
C07976=1179.276,282.791,-68.439,-176.947,7.589,148.559
C07977=1179.280,282.542,-68.410,-176.950,7.586,148.559
C07978=1179.284,282.294,-68.380,-176.952,7.584,148.559
C07979=1179.288,282.045,-68.351,-176.955,7.581,148.559
C07980=1179.293,281.798,-68.322,-176.958,7.578,148.559
C07981=1179.298,281.549,-68.294,-176.960,7.575,148.559
C07982=1179.301,281.301,-68.265,-176.963,7.573,148.559
C07983=1179.305,281.052,-68.235,-176.965,7.570,148.559
C07984=1179.310,280.804,-68.207,-176.968,7.567,148.559
C07985=1179.315,280.556,-68.178,-176.971,7.564,148.559
C07986=1179.319,280.307,-68.149,-176.974,7.561,148.559
C07987=1179.323,280.060,-68.120,-176.976,7.559,148.559
C07988=1179.328,279.811,-68.092,-176.978,7.556,148.559
C07989=1179.332,279.563,-68.062,-176.981,7.553,148.559
C07990=1179.336,279.314,-68.034,-176.984,7.550,148.559
C07991=1179.340,279.067,-68.005,-176.986,7.548,148.559
C07992=1179.345,278.818,-67.976,-176.989,7.545,148.559
C07993=1179.349,278.569,-67.947,-176.992,7.542,148.559
C07994=1179.353,278.322,-67.919,-176.994,7.539,148.559
C07995=1179.358,278.073,-67.890,-176.996,7.537,148.560
C07996=1179.362,277.824,-67.861,-176.999,7.534,148.560
C07997=1179.366,277.576,-67.833,-177.002,7.531,148.560
C07998=1179.371,277.328,-67.803,-177.005,7.528,148.560
C07999=1179.375,277.079,-67.775,-177.007,7.526,148.560
C08000=1179.379,276.831,-67.747,-177.009,7.523,148.560
C08001=1179.384,276.583,-67.718,-177.012,7.520,148.560
C08002=1179.387,276.335,-67.689,-177.015,7.517,148.560
C08003=1179.392,276.086,-67.661,-177.017,7.515,148.560
C08004=1179.397,275.838,-67.632,-177.020,7.512,148.560
C08005=1179.400,275.590,-67.603,-177.023,7.509,148.560
C08006=1179.405,275.341,-67.575,-177.025,7.506,148.560
C08007=1179.409,275.093,-67.547,-177.027,7.504,148.560
C08008=1179.414,274.845,-67.518,-177.030,7.501,148.560
C08009=1179.418,274.596,-67.489,-177.033,7.498,148.560
C08010=1179.422,274.348,-67.461,-177.036,7.495,148.560
C08011=1179.427,274.100,-67.433,-177.038,7.492,148.560
C08012=1179.431,273.851,-67.404,-177.041,7.489,148.560
C08013=1179.436,273.603,-67.375,-177.043,7.486,148.560
C08014=1179.440,273.355,-67.347,-177.047,7.484,148.561
C08015=1179.444,273.106,-67.318,-177.049,7.482,148.561
C08016=1179.448,272.858,-67.291,-177.051,7.479,148.561
C08017=1179.453,272.609,-67.262,-177.054,7.476,148.561
C08018=1179.457,272.361,-67.234,-177.056,7.474,148.561
C08019=1179.462,272.112,-67.205,-177.059,7.471,148.561
C08020=1179.466,271.865,-67.178,-177.062,7.468,148.561
C08021=1179.470,271.616,-67.148,-177.065,7.465,148.561
C08022=1179.475,271.368,-67.120,-177.067,7.462,148.561
C08023=1179.479,271.120,-67.092,-177.069,7.459,148.561
C08024=1179.484,270.872,-67.064,-177.072,7.457,148.561
C08025=1179.488,270.623,-67.035,-177.074,7.454,148.561
C08026=1179.492,270.375,-67.007,-177.077,7.451,148.561
C08027=1179.496,270.126,-66.979,-177.080,7.448,148.561
C08028=1179.501,269.878,-66.951,-177.083,7.445,148.562
C08029=1179.505,269.630,-66.923,-177.085,7.444,148.562
C08030=1179.510,269.381,-66.894,-177.088,7.441,148.562
C08031=1179.514,269.133,-66.866,-177.091,7.438,148.562
C08032=1179.518,268.885,-66.838,-177.093,7.435,148.562
C08033=1179.523,268.635,-66.810,-177.096,7.432,148.562
C08034=1179.527,268.388,-66.783,-177.098,7.430,148.562
C08035=1179.532,268.139,-66.754,-177.101,7.427,148.562
C08036=1179.536,267.891,-66.726,-177.103,7.424,148.562
C08037=1179.540,267.642,-66.698,-177.106,7.421,148.562
C08038=1179.545,267.394,-66.670,-177.109,7.418,148.562
C08039=1179.549,267.145,-66.641,-177.111,7.416,148.562
C08040=1179.553,266.898,-66.614,-177.114,7.414,148.563
C08041=1179.558,266.648,-66.586,-177.117,7.411,148.563
C08042=1179.562,266.400,-66.558,-177.119,7.408,148.563
C08043=1179.567,266.152,-66.530,-177.122,7.406,148.563
C08044=1179.570,265.904,-66.502,-177.124,7.403,148.563
C08045=1179.575,265.656,-66.474,-177.127,7.400,148.563
C08046=1179.579,265.406,-66.446,-177.129,7.397,148.563
C08047=1179.584,265.158,-66.418,-177.132,7.394,148.563
C08048=1179.589,264.910,-66.390,-177.135,7.393,148.563
C08049=1179.593,264.661,-66.363,-177.137,7.390,148.563
C08050=1179.597,264.413,-66.335,-177.140,7.387,148.563
C08051=1179.601,264.165,-66.307,-177.142,7.384,148.564
C08052=1179.605,263.917,-66.279,-177.145,7.381,148.564
C08053=1179.611,263.668,-66.251,-177.148,7.379,148.564
C08054=1179.615,263.419,-66.223,-177.150,7.376,148.564
C08055=1179.619,263.172,-66.195,-177.153,7.374,148.564
C08056=1179.623,262.922,-66.168,-177.156,7.371,148.564
C08057=1179.628,262.650,-66.138,-177.159,7.368,148.564
C08058=1179.633,262.376,-66.107,-177.161,7.365,148.564
C08059=1179.638,262.104,-66.077,-177.165,7.362,148.564
C08060=1179.643,261.830,-66.046,-177.167,7.359,148.565
C08061=1179.647,261.583,-66.018,-177.169,7.357,148.565
C08062=1179.651,261.333,-65.991,-177.172,7.354,148.565
C08063=1179.656,261.085,-65.963,-177.175,7.351,148.565
C08064=1179.660,260.837,-65.936,-177.177,7.349,148.565
C08065=1179.664,260.588,-65.908,-177.180,7.346,148.565
C08066=1179.669,260.340,-65.881,-177.183,7.343,148.565
C08067=1179.673,260.092,-65.853,-177.185,7.341,148.565
C08068=1179.678,259.843,-65.825,-177.188,7.338,148.565
C08069=1179.682,259.595,-65.797,-177.191,7.335,148.565
C08070=1179.687,259.346,-65.770,-177.193,7.333,148.566
C08071=1179.691,259.098,-65.742,-177.196,7.330,148.566
C08072=1179.695,258.849,-65.715,-177.199,7.327,148.566
C08073=1179.700,258.601,-65.687,-177.201,7.325,148.566
C08074=1179.704,258.353,-65.660,-177.204,7.322,148.566
C08075=1179.709,258.104,-65.633,-177.206,7.320,148.566
C08076=1179.713,257.856,-65.605,-177.209,7.317,148.566
C08077=1179.717,257.607,-65.578,-177.212,7.314,148.566
C08078=1179.722,257.359,-65.551,-177.214,7.312,148.566
C08079=1179.726,257.111,-65.523,-177.217,7.309,148.566
C08080=1179.730,256.862,-65.495,-177.220,7.307,148.567
C08081=1179.735,256.613,-65.468,-177.222,7.305,148.567
C08082=1179.739,256.365,-65.441,-177.225,7.302,148.567
C08083=1179.744,256.117,-65.414,-177.227,7.299,148.567
C08084=1179.748,255.867,-65.386,-177.230,7.296,148.567
C08085=1179.752,255.620,-65.358,-177.233,7.294,148.567
C08086=1179.757,255.371,-65.331,-177.235,7.292,148.567
C08087=1179.762,255.123,-65.304,-177.238,7.289,148.567
C08088=1179.766,254.874,-65.278,-177.240,7.287,148.568
C08089=1179.770,254.625,-65.250,-177.243,7.284,148.568
C08090=1179.774,254.377,-65.223,-177.246,7.281,148.568
C08091=1179.779,254.129,-65.195,-177.248,7.279,148.568
C08092=1179.783,253.880,-65.168,-177.251,7.276,148.568
C08093=1179.788,253.632,-65.141,-177.254,7.274,148.568
C08094=1179.792,253.383,-65.114,-177.256,7.271,148.568
C08095=1179.797,253.134,-65.087,-177.259,7.268,148.568
C08096=1179.800,252.887,-65.060,-177.261,7.266,148.569
C08097=1179.805,252.638,-65.033,-177.264,7.263,148.569
C08098=1179.810,252.390,-65.006,-177.267,7.261,148.569
C08099=1179.814,252.141,-64.979,-177.269,7.258,148.569
C08100=1179.818,251.892,-64.951,-177.272,7.255,148.569
C08101=1179.823,251.643,-64.924,-177.275,7.253,148.569
C08102=1179.827,251.395,-64.898,-177.277,7.250,148.569
C08103=1179.832,251.147,-64.870,-177.280,7.248,148.569
C08104=1179.836,250.898,-64.843,-177.283,7.246,148.570
C08105=1179.841,250.650,-64.816,-177.285,7.243,148.570
C08106=1179.846,250.401,-64.789,-177.288,7.240,148.570
C08107=1179.849,250.153,-64.763,-177.290,7.237,148.570
C08108=1179.854,249.905,-64.736,-177.293,7.236,148.570
C08109=1179.858,249.655,-64.708,-177.296,7.233,148.570
C08110=1179.863,249.407,-64.681,-177.298,7.230,148.570
C08111=1179.867,249.159,-64.655,-177.301,7.228,148.571
C08112=1179.871,248.910,-64.628,-177.303,7.226,148.571
C08113=1179.876,248.662,-64.601,-177.306,7.223,148.571
C08114=1179.880,248.414,-64.574,-177.309,7.220,148.571
C08115=1179.885,248.165,-64.547,-177.312,7.218,148.571
C08116=1179.890,247.916,-64.521,-177.314,7.215,148.571
C08117=1179.894,247.668,-64.494,-177.316,7.213,148.571
C08118=1179.898,247.419,-64.467,-177.320,7.210,148.572
C08119=1179.903,247.171,-64.440,-177.322,7.208,148.572
C08120=1179.907,246.923,-64.414,-177.325,7.205,148.572
C08121=1179.911,246.674,-64.387,-177.327,7.203,148.572
C08122=1179.916,246.425,-64.360,-177.330,7.200,148.572
C08123=1179.920,246.177,-64.334,-177.333,7.197,148.572
C08124=1179.925,245.928,-64.307,-177.335,7.195,148.573
C08125=1179.930,245.680,-64.280,-177.338,7.193,148.573
C08126=1179.934,245.432,-64.253,-177.340,7.190,148.573
C08127=1179.938,245.182,-64.227,-177.343,7.188,148.573
C08128=1179.942,244.934,-64.201,-177.346,7.186,148.573
C08129=1179.947,244.686,-64.173,-177.348,7.183,148.573
C08130=1179.952,244.437,-64.147,-177.351,7.181,148.574
C08131=1179.956,244.189,-64.121,-177.354,7.178,148.574
C08132=1179.961,243.940,-64.094,-177.356,7.176,148.574
C08133=1179.965,243.691,-64.068,-177.359,7.173,148.574
C08134=1179.969,243.443,-64.041,-177.361,7.171,148.574
C08135=1179.973,243.195,-64.014,-177.364,7.168,148.574
C08136=1179.978,242.945,-63.988,-177.367,7.166,148.574
C08137=1179.982,242.697,-63.961,-177.369,7.163,148.575
C08138=1179.987,242.449,-63.934,-177.373,7.160,148.575
C08139=1179.991,242.200,-63.909,-177.375,7.158,148.575
C08140=1179.996,241.951,-63.882,-177.378,7.155,148.575
C08141=1180.000,241.703,-63.856,-177.380,7.154,148.575
C08142=1180.005,241.454,-63.829,-177.383,7.151,148.575
C08143=1180.009,241.205,-63.803,-177.385,7.148,148.575
C08144=1180.014,240.957,-63.776,-177.388,7.146,148.576
C08145=1180.018,240.708,-63.750,-177.391,7.144,148.576
C08146=1180.022,240.460,-63.723,-177.394,7.141,148.576
C08147=1180.027,240.211,-63.697,-177.396,7.139,148.576
C08148=1180.031,239.962,-63.670,-177.399,7.136,148.576
C08149=1180.036,239.714,-63.645,-177.401,7.134,148.577
C08150=1180.040,239.466,-63.619,-177.404,7.131,148.577
C08151=1180.045,239.217,-63.592,-177.407,7.129,148.577
C08152=1180.049,238.969,-63.566,-177.409,7.126,148.577
C08153=1180.054,238.720,-63.539,-177.412,7.124,148.577
C08154=1180.058,238.471,-63.513,-177.415,7.122,148.578
C08155=1180.062,238.223,-63.487,-177.417,7.119,148.578
C08156=1180.067,237.973,-63.461,-177.420,7.117,148.578
C08157=1180.072,237.726,-63.435,-177.422,7.115,148.578
C08158=1180.076,237.477,-63.409,-177.425,7.112,148.578
C08159=1180.081,237.228,-63.383,-177.428,7.110,148.578
C08160=1180.085,236.980,-63.356,-177.430,7.108,148.578
C08161=1180.089,236.708,-63.328,-177.433,7.105,148.579
C08162=1180.094,236.436,-63.299,-177.436,7.102,148.579
C08163=1180.100,236.165,-63.271,-177.439,7.099,148.579
C08164=1180.104,235.894,-63.242,-177.442,7.097,148.579
C08165=1180.109,235.645,-63.216,-177.445,7.095,148.580
C08166=1180.113,235.396,-63.190,-177.447,7.092,148.580
C08167=1180.118,235.147,-63.164,-177.450,7.090,148.580
C08168=1180.121,234.899,-63.138,-177.453,7.087,148.580
C08169=1180.127,234.651,-63.112,-177.455,7.085,148.580
C08170=1180.131,234.402,-63.086,-177.458,7.083,148.580
C08171=1180.135,234.153,-63.061,-177.461,7.080,148.581
C08172=1180.139,233.905,-63.034,-177.463,7.078,148.581
C08173=1180.145,233.656,-63.008,-177.466,7.076,148.581
C08174=1180.149,233.408,-62.982,-177.468,7.073,148.581
C08175=1180.153,233.159,-62.957,-177.472,7.071,148.582
C08176=1180.158,232.910,-62.931,-177.474,7.069,148.582
C08177=1180.162,232.661,-62.905,-177.476,7.066,148.582
C08178=1180.167,232.413,-62.879,-177.479,7.064,148.582
C08179=1180.172,232.164,-62.853,-177.481,7.062,148.582
C08180=1180.176,231.916,-62.827,-177.485,7.059,148.582
C08181=1180.180,231.668,-62.801,-177.487,7.057,148.583
C08182=1180.185,231.419,-62.776,-177.490,7.054,148.583
C08183=1180.189,231.170,-62.750,-177.492,7.052,148.583
C08184=1180.194,230.921,-62.724,-177.495,7.050,148.583
C08185=1180.199,230.673,-62.698,-177.497,7.047,148.583
C08186=1180.203,230.424,-62.672,-177.501,7.045,148.584
C08187=1180.207,230.175,-62.647,-177.503,7.043,148.584
C08188=1180.211,229.926,-62.621,-177.506,7.041,148.584
C08189=1180.216,229.678,-62.596,-177.508,7.038,148.584
C08190=1180.220,229.429,-62.570,-177.511,7.036,148.584
C08191=1180.225,229.181,-62.544,-177.514,7.033,148.585
C08192=1180.229,228.933,-62.519,-177.516,7.031,148.585
C08193=1180.234,228.684,-62.493,-177.519,7.028,148.585
C08194=1180.238,228.434,-62.468,-177.522,7.026,148.585
C08195=1180.243,228.186,-62.443,-177.524,7.024,148.585
C08196=1180.248,227.937,-62.416,-177.527,7.022,148.586
C08197=1180.252,227.688,-62.390,-177.529,7.020,148.586
C08198=1180.257,227.440,-62.365,-177.533,7.017,148.586
C08199=1180.261,227.191,-62.339,-177.535,7.015,148.586
C08200=1180.265,226.943,-62.314,-177.537,7.013,148.587
C08201=1180.270,226.694,-62.288,-177.541,7.010,148.587
C08202=1180.275,226.445,-62.263,-177.543,7.008,148.587
C08203=1180.280,226.197,-62.238,-177.546,7.006,148.587
C08204=1180.284,225.948,-62.212,-177.548,7.003,148.587
C08205=1180.288,225.699,-62.186,-177.551,7.002,148.588
C08206=1180.292,225.452,-62.161,-177.554,6.999,148.588
C08207=1180.297,225.202,-62.136,-177.556,6.997,148.588
C08208=1180.301,224.953,-62.111,-177.559,6.994,148.588
C08209=1180.306,224.705,-62.085,-177.562,6.992,148.588
C08210=1180.310,224.456,-62.060,-177.564,6.990,148.589
C08211=1180.315,224.208,-62.035,-177.567,6.987,148.589
C08212=1180.319,223.959,-62.009,-177.570,6.986,148.589
C08213=1180.324,223.710,-61.983,-177.572,6.983,148.589
C08214=1180.329,223.461,-61.959,-177.575,6.981,148.590
C08215=1180.333,223.213,-61.933,-177.577,6.979,148.590
C08216=1180.338,222.964,-61.908,-177.580,6.976,148.590
C08217=1180.342,222.715,-61.883,-177.583,6.974,148.590
C08218=1180.346,222.467,-61.858,-177.585,6.972,148.590
C08219=1180.351,222.218,-61.833,-177.589,6.969,148.591
C08220=1180.356,221.970,-61.807,-177.591,6.967,148.591
C08221=1180.360,221.721,-61.782,-177.594,6.965,148.591
C08222=1180.364,221.471,-61.757,-177.596,6.962,148.591
C08223=1180.369,221.223,-61.731,-177.599,6.961,148.592
C08224=1180.373,220.974,-61.707,-177.602,6.958,148.592
C08225=1180.378,220.726,-61.681,-177.604,6.956,148.592
C08226=1180.382,220.477,-61.656,-177.607,6.954,148.592
C08227=1180.387,220.229,-61.631,-177.610,6.951,148.592
C08228=1180.392,219.979,-61.606,-177.612,6.949,148.593
C08229=1180.396,219.731,-61.581,-177.614,6.947,148.593
C08230=1180.400,219.482,-61.556,-177.618,6.945,148.593
C08231=1180.405,219.234,-61.531,-177.620,6.943,148.594
C08232=1180.410,218.984,-61.506,-177.623,6.940,148.594
C08233=1180.414,218.737,-61.481,-177.626,6.938,148.594
C08234=1180.418,218.487,-61.456,-177.628,6.936,148.594
C08235=1180.423,218.239,-61.430,-177.631,6.933,148.594
C08236=1180.428,217.990,-61.405,-177.634,6.931,148.595
C08237=1180.432,217.742,-61.381,-177.636,6.929,148.595
C08238=1180.436,217.492,-61.356,-177.639,6.927,148.595
C08239=1180.442,217.244,-61.331,-177.642,6.925,148.596
C08240=1180.446,216.996,-61.306,-177.644,6.923,148.596
C08241=1180.450,216.747,-61.281,-177.647,6.920,148.596
C08242=1180.455,216.498,-61.256,-177.649,6.918,148.596
C08243=1180.459,216.249,-61.231,-177.652,6.916,148.596
C08244=1180.464,216.001,-61.207,-177.655,6.914,148.597
C08245=1180.468,215.751,-61.182,-177.658,6.911,148.597
C08246=1180.473,215.503,-61.157,-177.660,6.910,148.597
C08247=1180.478,215.255,-61.132,-177.663,6.907,148.597
C08248=1180.482,215.005,-61.107,-177.666,6.905,148.598
C08249=1180.487,214.757,-61.083,-177.668,6.903,148.598
C08250=1180.491,214.508,-61.057,-177.671,6.900,148.598
C08251=1180.495,214.260,-61.033,-177.674,6.898,148.598
C08252=1180.500,214.011,-61.008,-177.676,6.897,148.599
C08253=1180.505,213.761,-60.983,-177.679,6.894,148.599
C08254=1180.509,213.514,-60.959,-177.682,6.892,148.599
C08255=1180.513,213.264,-60.934,-177.684,6.890,148.599
C08256=1180.518,213.016,-60.910,-177.687,6.887,148.600
C08257=1180.523,212.767,-60.885,-177.690,6.885,148.600
C08258=1180.527,212.518,-60.860,-177.692,6.883,148.600
C08259=1180.532,212.269,-60.836,-177.695,6.881,148.600
C08260=1180.536,212.021,-60.812,-177.698,6.879,148.601
C08261=1180.541,211.772,-60.786,-177.701,6.877,148.601
C08262=1180.546,211.523,-60.761,-177.703,6.875,148.601
C08263=1180.550,211.275,-60.737,-177.706,6.872,148.601
C08264=1180.555,211.025,-60.712,-177.709,6.870,148.602
C08265=1180.559,210.756,-60.686,-177.712,6.868,148.602
C08266=1180.564,210.485,-60.659,-177.714,6.866,148.602
C08267=1180.569,210.214,-60.633,-177.717,6.863,148.602
C08268=1180.574,209.944,-60.606,-177.720,6.861,148.603
C08269=1180.579,209.695,-60.582,-177.723,6.858,148.603
C08270=1180.583,209.446,-60.557,-177.725,6.856,148.603
C08271=1180.588,209.197,-60.532,-177.728,6.855,148.604
C08272=1180.593,208.949,-60.508,-177.731,6.853,148.604
C08273=1180.597,208.700,-60.484,-177.733,6.850,148.604
C08274=1180.602,208.451,-60.459,-177.736,6.848,148.604
C08275=1180.606,208.203,-60.435,-177.739,6.846,148.605
C08276=1180.611,207.954,-60.411,-177.742,6.844,148.605
C08277=1180.615,207.705,-60.386,-177.744,6.841,148.605
C08278=1180.619,207.456,-60.362,-177.747,6.840,148.605
C08279=1180.624,207.208,-60.337,-177.749,6.838,148.606
C08280=1180.629,206.959,-60.313,-177.752,6.835,148.606
C08281=1180.634,206.710,-60.289,-177.755,6.833,148.606
C08282=1180.638,206.461,-60.265,-177.758,6.831,148.607
C08283=1180.642,206.212,-60.241,-177.760,6.828,148.607
C08284=1180.648,205.964,-60.216,-177.763,6.827,148.607
C08285=1180.652,205.715,-60.192,-177.766,6.825,148.607
C08286=1180.656,205.466,-60.168,-177.768,6.823,148.608
C08287=1180.661,205.217,-60.144,-177.771,6.820,148.608
C08288=1180.666,204.968,-60.120,-177.774,6.818,148.608
C08289=1180.670,204.720,-60.096,-177.776,6.816,148.608
C08290=1180.675,204.471,-60.071,-177.779,6.814,148.609
C08291=1180.679,204.222,-60.046,-177.782,6.812,148.609
C08292=1180.684,203.973,-60.023,-177.784,6.810,148.609
C08293=1180.688,203.725,-59.999,-177.787,6.808,148.610
C08294=1180.693,203.476,-59.974,-177.789,6.806,148.610
C08295=1180.697,203.227,-59.950,-177.793,6.803,148.610
C08296=1180.702,202.978,-59.927,-177.795,6.802,148.610
C08297=1180.706,202.729,-59.902,-177.798,6.800,148.611
C08298=1180.711,202.481,-59.878,-177.800,6.798,148.611
C08299=1180.716,202.232,-59.854,-177.803,6.795,148.611
C08300=1180.720,201.983,-59.830,-177.806,6.793,148.612
C08301=1180.725,201.735,-59.806,-177.808,6.791,148.612
C08302=1180.729,201.485,-59.783,-177.811,6.789,148.612
C08303=1180.734,201.236,-59.758,-177.813,6.787,148.612
C08304=1180.739,200.987,-59.735,-177.817,6.785,148.613
C08305=1180.743,200.739,-59.710,-177.819,6.783,148.613
C08306=1180.747,200.490,-59.686,-177.822,6.781,148.613
C08307=1180.752,200.241,-59.663,-177.824,6.779,148.613
C08308=1180.756,199.993,-59.639,-177.827,6.777,148.614
C08309=1180.762,199.744,-59.615,-177.830,6.774,148.614
C08310=1180.766,199.495,-59.591,-177.832,6.773,148.614
C08311=1180.770,199.245,-59.567,-177.835,6.771,148.615
C08312=1180.775,198.997,-59.543,-177.838,6.769,148.615
C08313=1180.779,198.748,-59.520,-177.841,6.766,148.615
C08314=1180.784,198.500,-59.496,-177.843,6.764,148.615
C08315=1180.789,198.251,-59.472,-177.846,6.762,148.616
C08316=1180.793,198.002,-59.448,-177.848,6.761,148.616
C08317=1180.798,197.753,-59.424,-177.852,6.758,148.616
C08318=1180.803,197.504,-59.400,-177.854,6.756,148.617
C08319=1180.807,197.255,-59.377,-177.857,6.754,148.617
C08320=1180.812,197.007,-59.353,-177.859,6.752,148.617
C08321=1180.817,196.758,-59.329,-177.862,6.751,148.618
C08322=1180.821,196.509,-59.306,-177.865,6.748,148.618
C08323=1180.826,196.261,-59.282,-177.867,6.746,148.618
C08324=1180.830,196.011,-59.259,-177.870,6.744,148.618
C08325=1180.834,195.762,-59.235,-177.873,6.742,148.619
C08326=1180.839,195.513,-59.211,-177.875,6.740,148.619
C08327=1180.844,195.264,-59.187,-177.878,6.738,148.619
C08328=1180.848,195.016,-59.163,-177.881,6.736,148.620
C08329=1180.853,194.767,-59.140,-177.883,6.734,148.620
C08330=1180.857,194.518,-59.117,-177.886,6.732,148.620
C08331=1180.862,194.269,-59.093,-177.889,6.730,148.621
C08332=1180.866,194.020,-59.069,-177.891,6.728,148.621
C08333=1180.871,193.771,-59.046,-177.894,6.726,148.621
C08334=1180.876,193.522,-59.023,-177.897,6.724,148.621
C08335=1180.881,193.273,-58.999,-177.899,6.722,148.622
C08336=1180.885,193.025,-58.975,-177.902,6.720,148.622
C08337=1180.890,192.776,-58.952,-177.904,6.718,148.622
C08338=1180.895,192.528,-58.929,-177.907,6.716,148.623
C08339=1180.900,192.278,-58.905,-177.910,6.714,148.623
C08340=1180.903,192.030,-58.882,-177.913,6.712,148.623
C08341=1180.908,191.781,-58.859,-177.916,6.710,148.624
C08342=1180.913,191.532,-58.835,-177.918,6.708,148.624
C08343=1180.917,191.283,-58.812,-177.920,6.706,148.624
C08344=1180.922,191.034,-58.788,-177.923,6.704,148.624
C08345=1180.927,190.785,-58.765,-177.926,6.702,148.625
C08346=1180.931,190.536,-58.742,-177.929,6.700,148.625
C08347=1180.936,190.288,-58.718,-177.932,6.698,148.625
C08348=1180.940,190.039,-58.695,-177.934,6.696,148.626
C08349=1180.945,189.790,-58.672,-177.937,6.694,148.626
C08350=1180.949,189.541,-58.648,-177.939,6.693,148.626
C08351=1180.954,189.292,-58.625,-177.942,6.690,148.627
C08352=1180.959,189.043,-58.601,-177.945,6.688,148.627
C08353=1180.964,188.795,-58.578,-177.948,6.686,148.627
C08354=1180.968,188.546,-58.556,-177.950,6.684,148.627
C08355=1180.973,188.297,-58.532,-177.953,6.682,148.628
C08356=1180.977,188.048,-58.509,-177.955,6.681,148.628
C08357=1180.982,187.799,-58.486,-177.958,6.679,148.629
C08358=1180.987,187.550,-58.462,-177.961,6.676,148.629
C08359=1180.991,187.301,-58.440,-177.964,6.675,148.629
C08360=1180.995,187.052,-58.416,-177.967,6.673,148.630
C08361=1181.001,186.804,-58.393,-177.969,6.671,148.630
C08362=1181.005,186.555,-58.370,-177.971,6.669,148.630
C08363=1181.009,186.306,-58.347,-177.974,6.667,148.630
C08364=1181.014,186.057,-58.324,-177.977,6.665,148.631
C08365=1181.019,185.808,-58.300,-177.979,6.663,148.631
C08366=1181.023,185.558,-58.278,-177.983,6.661,148.631
C08367=1181.028,185.310,-58.255,-177.985,6.659,148.632
C08368=1181.033,185.061,-58.232,-177.988,6.657,148.632
C08369=1181.038,184.792,-58.207,-177.990,6.655,148.632
C08370=1181.043,184.522,-58.182,-177.993,6.653,148.633
C08371=1181.048,184.253,-58.157,-177.996,6.651,148.633
C08372=1181.052,183.983,-58.132,-177.999,6.649,148.634
C08373=1181.057,183.734,-58.110,-178.002,6.647,148.634
C08374=1181.062,183.485,-58.086,-178.005,6.645,148.634
C08375=1181.066,183.236,-58.063,-178.007,6.643,148.634
C08376=1181.071,182.987,-58.040,-178.010,6.641,148.635
C08377=1181.076,182.739,-58.017,-178.013,6.639,148.635
C08378=1181.080,182.489,-57.995,-178.015,6.637,148.636
C08379=1181.085,182.240,-57.972,-178.018,6.636,148.636
C08380=1181.089,181.991,-57.949,-178.021,6.634,148.636
C08381=1181.094,181.743,-57.926,-178.023,6.632,148.636
C08382=1181.099,181.493,-57.903,-178.026,6.630,148.637
C08383=1181.103,181.245,-57.881,-178.028,6.628,148.637
C08384=1181.108,180.996,-57.857,-178.031,6.626,148.637
C08385=1181.113,180.747,-57.836,-178.034,6.624,148.638
C08386=1181.118,180.498,-57.812,-178.037,6.622,148.638
C08387=1181.122,180.249,-57.789,-178.040,6.620,148.638
C08388=1181.127,180.000,-57.767,-178.042,6.619,148.639
C08389=1181.131,179.752,-57.744,-178.045,6.617,148.639
C08390=1181.136,179.503,-57.721,-178.048,6.615,148.640
C08391=1181.140,179.253,-57.699,-178.050,6.613,148.640
C08392=1181.145,179.004,-57.676,-178.052,6.611,148.640
C08393=1181.150,178.756,-57.654,-178.055,6.609,148.640
C08394=1181.154,178.507,-57.631,-178.058,6.607,148.641
C08395=1181.159,178.257,-57.608,-178.061,6.606,148.641
C08396=1181.164,178.009,-57.586,-178.063,6.604,148.642
C08397=1181.168,177.760,-57.563,-178.066,6.601,148.642
C08398=1181.173,177.511,-57.540,-178.069,6.600,148.642
C08399=1181.177,177.263,-57.518,-178.072,6.598,148.643
C08400=1181.182,177.013,-57.495,-178.074,6.596,148.643
C08401=1181.186,176.764,-57.472,-178.077,6.594,148.643
C08402=1181.192,176.515,-57.450,-178.080,6.592,148.644
C08403=1181.196,176.266,-57.427,-178.082,6.590,148.644
C08404=1181.200,176.017,-57.405,-178.085,6.589,148.644
C08405=1181.206,175.768,-57.383,-178.087,6.587,148.645
C08406=1181.210,175.519,-57.360,-178.090,6.585,148.645
C08407=1181.215,175.270,-57.338,-178.093,6.583,148.645
C08408=1181.219,175.022,-57.315,-178.095,6.581,148.646
C08409=1181.224,174.772,-57.293,-178.098,6.580,148.646
C08410=1181.228,174.523,-57.270,-178.101,6.578,148.646
C08411=1181.233,174.275,-57.248,-178.103,6.576,148.647
C08412=1181.238,174.025,-57.225,-178.106,6.574,148.647
C08413=1181.243,173.777,-57.203,-178.109,6.573,148.647
C08414=1181.247,173.528,-57.181,-178.111,6.571,148.648
C08415=1181.252,173.278,-57.158,-178.114,6.569,148.648
C08416=1181.257,173.030,-57.136,-178.117,6.567,148.649
C08417=1181.261,172.781,-57.114,-178.120,6.565,148.649
C08418=1181.267,172.532,-57.092,-178.123,6.563,148.649
C08419=1181.271,172.283,-57.069,-178.125,6.561,148.650
C08420=1181.275,172.034,-57.047,-178.128,6.559,148.650
C08421=1181.280,171.785,-57.025,-178.131,6.558,148.650
C08422=1181.285,171.535,-57.002,-178.133,6.555,148.650
C08423=1181.289,171.287,-56.980,-178.136,6.554,148.651
C08424=1181.293,171.038,-56.958,-178.138,6.552,148.651
C08425=1181.299,170.789,-56.936,-178.141,6.550,148.652
C08426=1181.303,170.540,-56.914,-178.144,6.548,148.652
C08427=1181.308,170.292,-56.891,-178.146,6.547,148.652
C08428=1181.312,170.042,-56.869,-178.149,6.545,148.653
C08429=1181.318,169.793,-56.847,-178.152,6.543,148.653
C08430=1181.322,169.544,-56.825,-178.154,6.541,148.653
C08431=1181.326,169.295,-56.803,-178.157,6.539,148.654
C08432=1181.331,169.046,-56.781,-178.160,6.538,148.654
C08433=1181.335,168.797,-56.758,-178.162,6.536,148.654
C08434=1181.341,168.548,-56.736,-178.165,6.534,148.655
C08435=1181.345,168.299,-56.714,-178.168,6.532,148.655
C08436=1181.350,168.050,-56.692,-178.170,6.531,148.656
C08437=1181.354,167.801,-56.670,-178.173,6.529,148.656
C08438=1181.359,167.553,-56.649,-178.176,6.527,148.656
C08439=1181.364,167.303,-56.626,-178.179,6.525,148.657
C08440=1181.369,167.054,-56.604,-178.181,6.523,148.657
C08441=1181.374,166.806,-56.583,-178.184,6.522,148.657
C08442=1181.378,166.556,-56.561,-178.187,6.520,148.658
C08443=1181.383,166.308,-56.539,-178.189,6.518,148.658
C08444=1181.387,166.058,-56.517,-178.192,6.516,148.659
C08445=1181.392,165.810,-56.495,-178.195,6.515,148.659
C08446=1181.396,165.560,-56.473,-178.197,6.513,148.659
C08447=1181.402,165.311,-56.451,-178.200,6.511,148.660
C08448=1181.406,165.062,-56.429,-178.203,6.509,148.660
C08449=1181.411,164.813,-56.407,-178.205,6.508,148.660
C08450=1181.415,164.564,-56.385,-178.208,6.506,148.661
C08451=1181.420,164.315,-56.363,-178.211,6.504,148.661
C08452=1181.425,164.067,-56.342,-178.213,6.502,148.661
C08453=1181.429,163.817,-56.320,-178.216,6.500,148.662
C08454=1181.434,163.569,-56.298,-178.219,6.499,148.662
C08455=1181.438,163.319,-56.276,-178.221,6.498,148.663
C08456=1181.443,163.071,-56.254,-178.224,6.496,148.663
C08457=1181.448,162.821,-56.232,-178.226,6.494,148.663
C08458=1181.453,162.572,-56.211,-178.229,6.492,148.664
C08459=1181.458,162.324,-56.190,-178.232,6.491,148.664
C08460=1181.462,162.074,-56.168,-178.234,6.489,148.664
C08461=1181.467,161.826,-56.146,-178.237,6.487,148.665
C08462=1181.471,161.576,-56.124,-178.240,6.485,148.665
C08463=1181.476,161.328,-56.102,-178.242,6.484,148.666
C08464=1181.481,161.078,-56.081,-178.245,6.482,148.666
C08465=1181.485,160.829,-56.059,-178.248,6.480,148.667
C08466=1181.490,160.580,-56.037,-178.251,6.479,148.667
C08467=1181.495,160.332,-56.016,-178.254,6.477,148.667
C08468=1181.500,160.082,-55.994,-178.256,6.475,148.668
C08469=1181.505,159.833,-55.973,-178.259,6.473,148.668
C08470=1181.509,159.584,-55.951,-178.262,6.472,148.668
C08471=1181.514,159.335,-55.929,-178.264,6.470,148.669
C08472=1181.518,159.086,-55.909,-178.267,6.468,148.669
C08473=1181.523,158.817,-55.885,-178.270,6.466,148.670
C08474=1181.528,158.548,-55.862,-178.272,6.464,148.670
C08475=1181.534,158.279,-55.838,-178.276,6.463,148.671
C08476=1181.538,158.011,-55.815,-178.278,6.461,148.671
C08477=1181.543,157.761,-55.794,-178.281,6.460,148.671
C08478=1181.548,157.513,-55.772,-178.284,6.458,148.672
C08479=1181.553,157.263,-55.751,-178.286,6.456,148.672
C08480=1181.557,157.014,-55.729,-178.289,6.454,148.672
C08481=1181.562,156.765,-55.708,-178.292,6.452,148.673
C08482=1181.567,156.515,-55.686,-178.294,6.451,148.673
C08483=1181.571,156.267,-55.665,-178.297,6.449,148.673
C08484=1181.576,156.018,-55.644,-178.300,6.447,148.674
C08485=1181.581,155.769,-55.623,-178.302,6.445,148.674
C08486=1181.585,155.520,-55.600,-178.305,6.444,148.675
C08487=1181.591,155.271,-55.579,-178.307,6.443,148.675
C08488=1181.595,155.022,-55.558,-178.310,6.441,148.676
C08489=1181.600,154.773,-55.537,-178.313,6.440,148.676
C08490=1181.604,154.524,-55.515,-178.316,6.438,148.676
C08491=1181.609,154.274,-55.494,-178.318,6.436,148.677
C08492=1181.614,154.026,-55.473,-178.321,6.434,148.677
C08493=1181.619,153.777,-55.452,-178.324,6.432,148.677
C08494=1181.623,153.528,-55.430,-178.326,6.431,148.678
C08495=1181.628,153.278,-55.409,-178.329,6.429,148.678
C08496=1181.633,153.029,-55.388,-178.332,6.427,148.679
C08497=1181.637,152.781,-55.367,-178.334,6.426,148.679
C08498=1181.643,152.531,-55.346,-178.337,6.424,148.679
C08499=1181.647,152.282,-55.324,-178.340,6.423,148.680
C08500=1181.652,152.033,-55.303,-178.342,6.421,148.680
C08501=1181.656,151.784,-55.282,-178.345,6.420,148.681
C08502=1181.661,151.535,-55.261,-178.348,6.418,148.681
C08503=1181.666,151.286,-55.240,-178.351,6.416,148.682
C08504=1181.670,151.037,-55.219,-178.353,6.414,148.682
C08505=1181.675,150.788,-55.198,-178.356,6.412,148.682
C08506=1181.680,150.538,-55.177,-178.358,6.412,148.683
C08507=1181.684,150.290,-55.156,-178.361,6.410,148.683
C08508=1181.690,150.041,-55.135,-178.363,6.408,148.683
C08509=1181.695,149.792,-55.114,-178.367,6.407,148.684
C08510=1181.698,149.543,-55.092,-178.369,6.405,148.684
C08511=1181.704,149.293,-55.071,-178.372,6.403,148.685
C08512=1181.708,149.044,-55.051,-178.375,6.401,148.685
C08513=1181.713,148.795,-55.030,-178.377,6.400,148.686
C08514=1181.718,148.546,-55.008,-178.379,6.399,148.686
C08515=1181.722,148.297,-54.988,-178.382,6.397,148.686
C08516=1181.728,148.048,-54.967,-178.385,6.395,148.687
C08517=1181.731,147.799,-54.946,-178.388,6.394,148.687
C08518=1181.736,147.550,-54.925,-178.391,6.392,148.688
C08519=1181.741,147.301,-54.904,-178.393,6.390,148.688
C08520=1181.746,147.052,-54.883,-178.396,6.388,148.688
C08521=1181.751,146.802,-54.862,-178.398,6.387,148.689
C08522=1181.756,146.553,-54.842,-178.401,6.386,148.689
C08523=1181.761,146.304,-54.821,-178.404,6.384,148.690
C08524=1181.765,146.056,-54.800,-178.406,6.382,148.690
C08525=1181.770,145.807,-54.779,-178.409,6.381,148.691
C08526=1181.774,145.558,-54.759,-178.412,6.379,148.691
C08527=1181.780,145.308,-54.738,-178.415,6.377,148.691
C08528=1181.783,145.059,-54.717,-178.417,6.376,148.692
C08529=1181.789,144.810,-54.696,-178.420,6.375,148.692
C08530=1181.793,144.561,-54.676,-178.422,6.373,148.693
C08531=1181.798,144.311,-54.655,-178.425,6.371,148.693
C08532=1181.803,144.062,-54.634,-178.428,6.370,148.694
C08533=1181.808,143.813,-54.613,-178.431,6.368,148.694
C08534=1181.812,143.565,-54.592,-178.433,6.367,148.694
C08535=1181.817,143.316,-54.571,-178.436,6.365,148.695
C08536=1181.822,143.067,-54.551,-178.438,6.363,148.695
C08537=1181.827,142.817,-54.530,-178.441,6.362,148.695
C08538=1181.831,142.568,-54.510,-178.444,6.360,148.696
C08539=1181.836,142.319,-54.489,-178.447,6.358,148.696
C08540=1181.841,142.070,-54.468,-178.449,6.358,148.697
C08541=1181.845,141.821,-54.448,-178.452,6.356,148.697
C08542=1181.851,141.571,-54.428,-178.454,6.354,148.698
C08543=1181.855,141.322,-54.407,-178.457,6.352,148.698
C08544=1181.860,141.073,-54.387,-178.460,6.351,148.699
C08545=1181.865,140.824,-54.366,-178.462,6.350,148.699
C08546=1181.869,140.575,-54.345,-178.465,6.348,148.699
C08547=1181.874,140.326,-54.325,-178.468,6.346,148.700
C08548=1181.879,140.077,-54.304,-178.470,6.345,148.700
C08549=1181.883,139.828,-54.284,-178.473,6.343,148.701
C08550=1181.888,139.579,-54.263,-178.476,6.342,148.701
C08551=1181.893,139.330,-54.242,-178.478,6.341,148.702
C08552=1181.898,139.080,-54.223,-178.481,6.339,148.702
C08553=1181.902,138.831,-54.202,-178.484,6.337,148.702
C08554=1181.907,138.582,-54.181,-178.487,6.335,148.703
C08555=1181.912,138.333,-54.161,-178.489,6.334,148.703
C08556=1181.916,138.084,-54.141,-178.492,6.333,148.704
C08557=1181.921,137.835,-54.120,-178.495,6.331,148.704
C08558=1181.926,137.585,-54.100,-178.497,6.329,148.704
C08559=1181.930,137.336,-54.080,-178.500,6.328,148.705
C08560=1181.936,137.087,-54.059,-178.502,6.327,148.705
C08561=1181.941,136.839,-54.039,-178.505,6.325,148.706
C08562=1181.945,136.589,-54.019,-178.508,6.324,148.706
C08563=1181.950,136.340,-53.999,-178.511,6.322,148.707
C08564=1181.955,136.091,-53.978,-178.513,6.320,148.707
C08565=1181.959,135.842,-53.957,-178.515,6.319,148.707
C08566=1181.964,135.593,-53.938,-178.519,6.318,148.708
C08567=1181.969,135.344,-53.917,-178.521,6.316,148.708
C08568=1181.973,135.095,-53.897,-178.524,6.314,148.709
C08569=1181.979,134.845,-53.877,-178.526,6.313,148.709
C08570=1181.983,134.596,-53.856,-178.529,6.312,148.710
C08571=1181.988,134.348,-53.836,-178.532,6.310,148.710
C08572=1181.993,134.098,-53.817,-178.535,6.308,148.711
C08573=1181.997,133.849,-53.796,-178.537,6.307,148.711
C08574=1182.003,133.599,-53.776,-178.540,6.306,148.711
C08575=1182.007,133.350,-53.756,-178.543,6.304,148.712
C08576=1182.012,133.101,-53.735,-178.545,6.303,148.712
C08577=1182.016,132.833,-53.714,-178.548,6.301,148.713
C08578=1182.022,132.564,-53.693,-178.551,6.299,148.713
C08579=1182.027,132.296,-53.671,-178.554,6.298,148.714
C08580=1182.032,132.027,-53.649,-178.557,6.296,148.714
C08581=1182.037,131.778,-53.629,-178.559,6.295,148.715
C08582=1182.042,131.529,-53.609,-178.562,6.294,148.715
C08583=1182.047,131.280,-53.589,-178.565,6.292,148.716
C08584=1182.051,131.030,-53.569,-178.567,6.290,148.716
C08585=1182.056,130.781,-53.549,-178.569,6.289,148.716
C08586=1182.061,130.532,-53.529,-178.573,6.288,148.717
C08587=1182.066,130.283,-53.508,-178.575,6.286,148.717
C08588=1182.071,130.034,-53.489,-178.578,6.284,148.718
C08589=1182.076,129.785,-53.469,-178.580,6.283,148.718
C08590=1182.080,129.535,-53.449,-178.583,6.282,148.719
C08591=1182.085,129.286,-53.429,-178.586,6.280,148.719
C08592=1182.090,129.037,-53.409,-178.589,6.278,148.720
C08593=1182.095,128.788,-53.390,-178.591,6.278,148.720
C08594=1182.099,128.539,-53.369,-178.594,6.276,148.721
C08595=1182.104,128.289,-53.350,-178.597,6.274,148.721
C08596=1182.108,128.040,-53.329,-178.599,6.273,148.721
C08597=1182.114,127.792,-53.310,-178.602,6.272,148.722
C08598=1182.118,127.542,-53.290,-178.605,6.270,148.722
C08599=1182.123,127.293,-53.270,-178.607,6.269,148.723
C08600=1182.128,127.043,-53.250,-178.610,6.268,148.723
C08601=1182.133,126.795,-53.231,-178.612,6.266,148.724
C08602=1182.137,126.546,-53.211,-178.615,6.265,148.724
C08603=1182.142,126.296,-53.191,-178.618,6.263,148.725
C08604=1182.148,126.047,-53.172,-178.620,6.262,148.725
C08605=1182.152,125.798,-53.151,-178.623,6.260,148.725
C08606=1182.157,125.549,-53.132,-178.626,6.259,148.726
C08607=1182.161,125.299,-53.112,-178.628,6.258,148.727
C08608=1182.167,125.050,-53.093,-178.631,6.256,148.727
C08609=1182.170,124.802,-53.073,-178.634,6.254,148.727
C08610=1182.175,124.552,-53.053,-178.637,6.253,148.728
C08611=1182.181,124.303,-53.034,-178.639,6.252,148.728
C08612=1182.185,124.054,-53.014,-178.642,6.250,148.729
C08613=1182.190,123.805,-52.994,-178.645,6.249,148.729
C08614=1182.195,123.556,-52.975,-178.647,6.248,148.730
C08615=1182.200,123.306,-52.955,-178.650,6.246,148.730
C08616=1182.205,123.057,-52.935,-178.652,6.244,148.731
C08617=1182.210,122.808,-52.916,-178.655,6.244,148.731
C08618=1182.214,122.559,-52.896,-178.658,6.242,148.732
C08619=1182.218,122.310,-52.877,-178.660,6.240,148.732
C08620=1182.224,122.061,-52.857,-178.663,6.240,148.733
C08621=1182.228,121.811,-52.838,-178.666,6.238,148.733
C08622=1182.233,121.562,-52.818,-178.668,6.236,148.733
C08623=1182.239,121.313,-52.799,-178.671,6.235,148.734
C08624=1182.243,121.063,-52.780,-178.674,6.234,148.734
C08625=1182.247,120.814,-52.760,-178.676,6.232,148.735
C08626=1182.253,120.565,-52.741,-178.679,6.230,148.735
C08627=1182.257,120.316,-52.720,-178.682,6.230,148.736
C08628=1182.262,120.066,-52.701,-178.684,6.228,148.736
C08629=1182.266,119.818,-52.682,-178.687,6.226,148.737
C08630=1182.271,119.568,-52.662,-178.689,6.226,148.737
C08631=1182.277,119.319,-52.643,-178.693,6.224,148.738
C08632=1182.281,119.070,-52.623,-178.695,6.222,148.738
C08633=1182.285,118.821,-52.604,-178.697,6.221,148.739
C08634=1182.291,118.572,-52.585,-178.701,6.220,148.739
C08635=1182.295,118.322,-52.565,-178.703,6.218,148.740
C08636=1182.301,118.073,-52.546,-178.705,6.217,148.740
C08637=1182.305,117.824,-52.527,-178.709,6.216,148.741
C08638=1182.310,117.575,-52.508,-178.711,6.214,148.741
C08639=1182.315,117.326,-52.488,-178.713,6.213,148.741
C08640=1182.320,117.075,-52.469,-178.716,6.212,148.742
C08641=1182.324,116.827,-52.451,-178.719,6.211,148.742
C08642=1182.329,116.577,-52.431,-178.721,6.209,148.743
C08643=1182.335,116.328,-52.412,-178.724,6.208,148.743
C08644=1182.339,116.079,-52.392,-178.727,6.207,148.744
C08645=1182.344,115.830,-52.373,-178.729,6.205,148.744
C08646=1182.349,115.581,-52.354,-178.732,6.204,148.745
C08647=1182.353,115.332,-52.335,-178.735,6.203,148.745
C08648=1182.358,115.083,-52.315,-178.737,6.201,148.746
C08649=1182.364,114.833,-52.297,-178.740,6.199,148.746
C08650=1182.368,114.584,-52.278,-178.743,6.199,148.747
C08651=1182.373,114.335,-52.258,-178.745,6.197,148.747
C08652=1182.378,114.085,-52.239,-178.748,6.195,148.748
C08653=1182.382,113.837,-52.220,-178.751,6.195,148.748
C08654=1182.387,113.587,-52.201,-178.753,6.193,148.749
C08655=1182.392,113.338,-52.182,-178.756,6.192,148.749
C08656=1182.397,113.089,-52.163,-178.759,6.191,148.750
C08657=1182.402,112.840,-52.143,-178.762,6.189,148.750
C08658=1182.406,112.591,-52.124,-178.764,6.188,148.750
C08659=1182.412,112.341,-52.106,-178.767,6.187,148.751
C08660=1182.416,112.092,-52.087,-178.770,6.185,148.751
C08661=1182.421,111.843,-52.067,-178.772,6.184,148.752
C08662=1182.425,111.593,-52.049,-178.775,6.183,148.753
C08663=1182.431,111.344,-52.030,-178.777,6.182,148.753
C08664=1182.435,111.095,-52.010,-178.780,6.180,148.753
C08665=1182.440,110.846,-51.991,-178.783,6.179,148.754
C08666=1182.445,110.596,-51.972,-178.785,6.178,148.754
C08667=1182.450,110.347,-51.954,-178.788,6.176,148.755
C08668=1182.455,110.098,-51.934,-178.790,6.176,148.755
C08669=1182.459,109.849,-51.916,-178.793,6.174,148.756
C08670=1182.465,109.600,-51.897,-178.796,6.172,148.756
C08671=1182.469,109.350,-51.878,-178.798,6.171,148.757
C08672=1182.474,109.101,-51.859,-178.801,6.170,148.757
C08673=1182.478,108.852,-51.840,-178.804,6.169,148.758
C08674=1182.484,108.602,-51.822,-178.806,6.167,148.758
C08675=1182.489,108.354,-51.803,-178.809,6.166,148.759
C08676=1182.493,108.104,-51.784,-178.812,6.165,148.759
C08677=1182.498,107.855,-51.765,-178.814,6.163,148.760
C08678=1182.502,107.606,-51.746,-178.817,6.162,148.760
C08679=1182.508,107.356,-51.728,-178.820,6.161,148.761
C08680=1182.513,107.108,-51.709,-178.822,6.159,148.761
C08681=1182.518,106.838,-51.688,-178.825,6.159,148.762
C08682=1182.523,106.570,-51.669,-178.828,6.157,148.762
C08683=1182.528,106.302,-51.648,-178.831,6.156,148.763
C08684=1182.534,106.033,-51.628,-178.834,6.154,148.763
C08685=1182.538,105.784,-51.609,-178.836,6.153,148.764
C08686=1182.543,105.535,-51.591,-178.839,6.152,148.764
C08687=1182.548,105.286,-51.572,-178.841,6.151,148.765
C08688=1182.553,105.036,-51.554,-178.844,6.149,148.765
C08689=1182.557,104.788,-51.535,-178.847,6.148,148.766
C08690=1182.562,104.538,-51.516,-178.850,6.147,148.766
C08691=1182.567,104.288,-51.498,-178.852,6.145,148.767
C08692=1182.573,104.040,-51.479,-178.855,6.144,148.767
C08693=1182.577,103.790,-51.460,-178.858,6.143,148.768
C08694=1182.582,103.541,-51.442,-178.860,6.142,148.768
C08695=1182.587,103.292,-51.423,-178.863,6.140,148.769
C08696=1182.592,103.042,-51.405,-178.866,6.139,148.769
C08697=1182.596,102.793,-51.386,-178.868,6.138,148.770
C08698=1182.601,102.544,-51.368,-178.871,6.137,148.770
C08699=1182.606,102.294,-51.349,-178.873,6.136,148.771
C08700=1182.611,102.045,-51.331,-178.876,6.134,148.771
C08701=1182.616,101.796,-51.313,-178.879,6.134,148.772
C08702=1182.621,101.547,-51.294,-178.881,6.132,148.772
C08703=1182.625,101.297,-51.275,-178.884,6.131,148.773
C08704=1182.630,101.048,-51.257,-178.887,6.130,148.773
C08705=1182.635,100.799,-51.239,-178.889,6.128,148.774
C08706=1182.640,100.549,-51.220,-178.892,6.127,148.774
C08707=1182.645,100.300,-51.201,-178.895,6.126,148.775
C08708=1182.650,100.051,-51.183,-178.897,6.125,148.775
C08709=1182.655,99.802,-51.165,-178.900,6.123,148.776
C08710=1182.660,99.552,-51.146,-178.902,6.122,148.776
C08711=1182.664,99.303,-51.128,-178.905,6.121,148.777
C08712=1182.669,99.054,-51.110,-178.907,6.120,148.777
C08713=1182.674,98.805,-51.092,-178.911,6.119,148.778
C08714=1182.678,98.555,-51.073,-178.913,6.118,148.778
C08715=1182.684,98.305,-51.055,-178.916,6.116,148.779
C08716=1182.689,98.057,-51.036,-178.918,6.116,148.779
C08717=1182.694,97.808,-51.018,-178.921,6.114,148.780
C08718=1182.698,97.559,-51.000,-178.924,6.112,148.781
C08719=1182.703,97.309,-50.982,-178.926,6.112,148.781
C08720=1182.708,97.060,-50.964,-178.929,6.110,148.782
C08721=1182.713,96.810,-50.945,-178.931,6.109,148.782
C08722=1182.718,96.561,-50.927,-178.934,6.108,148.782
C08723=1182.723,96.312,-50.909,-178.937,6.107,148.783
C08724=1182.727,96.062,-50.890,-178.940,6.105,148.783
C08725=1182.732,95.813,-50.872,-178.942,6.105,148.784
C08726=1182.737,95.564,-50.854,-178.945,6.103,148.785
C08727=1182.742,95.315,-50.836,-178.947,6.102,148.785
C08728=1182.747,95.066,-50.818,-178.950,6.101,148.786
C08729=1182.752,94.816,-50.800,-178.952,6.100,148.786
C08730=1182.757,94.566,-50.781,-178.956,6.098,148.787
C08731=1182.762,94.317,-50.763,-178.958,6.097,148.787
C08732=1182.767,94.068,-50.745,-178.961,6.096,148.788
C08733=1182.772,93.819,-50.727,-178.963,6.095,148.788
C08734=1182.776,93.570,-50.709,-178.966,6.094,148.789
C08735=1182.781,93.320,-50.692,-178.968,6.093,148.789
C08736=1182.786,93.071,-50.673,-178.971,6.091,148.790
C08737=1182.791,92.821,-50.655,-178.974,6.091,148.790
C08738=1182.795,92.572,-50.637,-178.976,6.089,148.791
C08739=1182.800,92.323,-50.619,-178.979,6.088,148.791
C08740=1182.805,92.074,-50.601,-178.982,6.087,148.792
C08741=1182.810,91.825,-50.583,-178.984,6.086,148.792
C08742=1182.815,91.576,-50.565,-178.987,6.084,148.793
C08743=1182.820,91.326,-50.547,-178.990,6.084,148.793
C08744=1182.824,91.076,-50.529,-178.992,6.082,148.794
C08745=1182.830,90.827,-50.512,-178.995,6.081,148.794
C08746=1182.834,90.578,-50.494,-178.998,6.080,148.795
C08747=1182.839,90.328,-50.476,-179.000,6.079,148.795
C08748=1182.844,90.079,-50.458,-179.003,6.078,148.796
C08749=1182.849,89.830,-50.440,-179.005,6.077,148.796
C08750=1182.854,89.581,-50.422,-179.008,6.075,148.797
C08751=1182.859,89.332,-50.404,-179.011,6.074,148.798
C08752=1182.864,89.082,-50.387,-179.013,6.074,148.798
C08753=1182.869,88.833,-50.369,-179.016,6.072,148.799
C08754=1182.874,88.584,-50.351,-179.019,6.072,148.799
C08755=1182.879,88.334,-50.333,-179.021,6.070,148.800
C08756=1182.884,88.085,-50.315,-179.023,6.069,148.800
C08757=1182.888,87.836,-50.298,-179.027,6.068,148.801
C08758=1182.893,87.586,-50.280,-179.029,6.067,148.801
C08759=1182.898,87.337,-50.262,-179.032,6.065,148.802
C08760=1182.903,87.087,-50.244,-179.034,6.064,148.802
C08761=1182.908,86.838,-50.226,-179.037,6.063,148.803
C08762=1182.913,86.588,-50.208,-179.039,6.062,148.803
C08763=1182.918,86.339,-50.190,-179.043,6.061,148.804
C08764=1182.922,86.090,-50.172,-179.045,6.060,148.804
C08765=1182.927,85.841,-50.156,-179.047,6.059,148.805
C08766=1182.932,85.591,-50.138,-179.050,6.058,148.805
C08767=1182.937,85.342,-50.120,-179.053,6.057,148.806
C08768=1182.942,85.092,-50.103,-179.055,6.055,148.807
C08769=1182.947,84.843,-50.085,-179.058,6.055,148.807
C08770=1182.952,84.594,-50.067,-179.061,6.053,148.808
C08771=1182.956,84.345,-50.050,-179.063,6.053,148.808
C08772=1182.961,84.095,-50.032,-179.066,6.051,148.809
C08773=1182.966,83.846,-50.015,-179.069,6.050,148.809
C08774=1182.971,83.597,-49.997,-179.071,6.049,148.810
C08775=1182.976,83.347,-49.979,-179.074,6.048,148.810
C08776=1182.981,83.098,-49.962,-179.076,6.047,148.811
C08777=1182.986,82.849,-49.944,-179.079,6.045,148.811
C08778=1182.991,82.600,-49.927,-179.082,6.045,148.812
C08779=1182.996,82.350,-49.909,-179.084,6.043,148.812
C08780=1183.001,82.102,-49.892,-179.087,6.043,148.813
C08781=1183.006,81.852,-49.875,-179.089,6.042,148.813
C08782=1183.011,81.603,-49.857,-179.092,6.040,148.814
C08783=1183.016,81.353,-49.839,-179.094,6.040,148.814
C08784=1183.020,81.104,-49.822,-179.098,6.038,148.815
C08785=1183.025,80.835,-49.803,-179.100,6.038,148.816
C08786=1183.031,80.566,-49.785,-179.103,6.036,148.816
C08787=1183.037,80.299,-49.765,-179.106,6.035,148.817
C08788=1183.042,80.030,-49.747,-179.109,6.034,148.817
C08789=1183.046,79.781,-49.729,-179.112,6.032,148.818
C08790=1183.051,79.531,-49.712,-179.114,6.032,148.819
C08791=1183.056,79.282,-49.694,-179.116,6.031,148.819
C08792=1183.061,79.032,-49.677,-179.119,6.030,148.820
C08793=1183.066,78.783,-49.660,-179.122,6.029,148.820
C08794=1183.071,78.534,-49.643,-179.125,6.027,148.821
C08795=1183.076,78.285,-49.626,-179.127,6.026,148.821
C08796=1183.081,78.035,-49.608,-179.130,6.026,148.822
C08797=1183.086,77.786,-49.591,-179.132,6.024,148.822
C08798=1183.091,77.536,-49.574,-179.135,6.024,148.823
C08799=1183.095,77.287,-49.556,-179.138,6.022,148.823
C08800=1183.100,77.038,-49.539,-179.140,6.021,148.824
C08801=1183.105,76.788,-49.522,-179.142,6.020,148.824
C08802=1183.111,76.539,-49.505,-179.146,6.019,148.825
C08803=1183.115,76.290,-49.488,-179.148,6.018,148.825
C08804=1183.120,76.040,-49.471,-179.151,6.017,148.826
C08805=1183.125,75.791,-49.453,-179.153,6.016,148.827
C08806=1183.130,75.541,-49.436,-179.156,6.015,148.827
C08807=1183.135,75.292,-49.419,-179.159,6.014,148.828
C08808=1183.140,75.043,-49.402,-179.161,6.013,148.828
C08809=1183.145,74.794,-49.384,-179.164,6.011,148.829
C08810=1183.149,74.544,-49.368,-179.166,6.011,148.829
C08811=1183.154,74.295,-49.350,-179.169,6.010,148.830
C08812=1183.159,74.045,-49.333,-179.172,6.009,148.830
C08813=1183.165,73.796,-49.316,-179.174,6.008,148.831
C08814=1183.169,73.547,-49.299,-179.177,6.007,148.832
C08815=1183.174,73.297,-49.282,-179.179,6.006,148.832
C08816=1183.179,73.048,-49.265,-179.182,6.005,148.833
C08817=1183.184,72.798,-49.248,-179.185,6.004,148.833
C08818=1183.190,72.549,-49.231,-179.187,6.003,148.834
C08819=1183.194,72.300,-49.214,-179.190,6.002,148.834
C08820=1183.199,72.050,-49.197,-179.193,6.001,148.835
C08821=1183.203,71.801,-49.179,-179.195,6.000,148.835
C08822=1183.208,71.552,-49.163,-179.197,5.999,148.836
C08823=1183.214,71.303,-49.146,-179.201,5.998,148.837
C08824=1183.218,71.053,-49.129,-179.203,5.997,148.837
C08825=1183.223,70.803,-49.112,-179.205,5.996,148.838
C08826=1183.228,70.554,-49.095,-179.208,5.995,148.838
C08827=1183.234,70.305,-49.078,-179.211,5.994,148.839
C08828=1183.238,70.055,-49.062,-179.213,5.993,148.839
C08829=1183.243,69.806,-49.044,-179.216,5.992,148.840
C08830=1183.248,69.557,-49.027,-179.219,5.991,148.840
C08831=1183.253,69.308,-49.011,-179.222,5.990,148.841
C08832=1183.258,69.058,-48.993,-179.224,5.989,148.842
C08833=1183.262,68.809,-48.977,-179.226,5.988,148.842
C08834=1183.268,68.559,-48.960,-179.229,5.987,148.843
C08835=1183.273,68.310,-48.943,-179.232,5.986,148.843
C08836=1183.277,68.060,-48.926,-179.234,5.985,148.844
C08837=1183.282,67.811,-48.909,-179.237,5.984,148.844
C08838=1183.287,67.562,-48.893,-179.240,5.983,148.845
C08839=1183.293,67.312,-48.876,-179.242,5.982,148.845
C08840=1183.297,67.063,-48.859,-179.245,5.981,148.846
C08841=1183.302,66.814,-48.843,-179.248,5.980,148.847
C08842=1183.307,66.564,-48.825,-179.250,5.980,148.847
C08843=1183.312,66.315,-48.809,-179.253,5.978,148.848
C08844=1183.317,66.066,-48.792,-179.255,5.977,148.848
C08845=1183.322,65.816,-48.775,-179.258,5.977,148.849
C08846=1183.327,65.566,-48.759,-179.260,5.975,148.849
C08847=1183.332,65.318,-48.742,-179.263,5.975,148.850
C08848=1183.337,65.067,-48.726,-179.265,5.974,148.850
C08849=1183.342,64.818,-48.709,-179.268,5.972,148.851
C08850=1183.347,64.569,-48.693,-179.271,5.972,148.852
C08851=1183.351,64.320,-48.676,-179.273,5.971,148.852
C08852=1183.357,64.070,-48.659,-179.276,5.970,148.853
C08853=1183.362,63.821,-48.642,-179.279,5.969,148.853
C08854=1183.366,63.571,-48.626,-179.281,5.968,148.854
C08855=1183.371,63.322,-48.609,-179.283,5.967,148.854
C08856=1183.377,63.072,-48.593,-179.287,5.966,148.855
C08857=1183.381,62.823,-48.576,-179.289,5.965,148.856
C08858=1183.386,62.574,-48.560,-179.291,5.964,148.856
C08859=1183.391,62.325,-48.543,-179.295,5.963,148.857
C08860=1183.396,62.075,-48.526,-179.297,5.962,148.857
C08861=1183.401,61.826,-48.510,-179.299,5.962,148.858
C08862=1183.406,61.576,-48.494,-179.302,5.960,148.858
C08863=1183.411,61.327,-48.477,-179.305,5.960,148.859
C08864=1183.416,61.077,-48.460,-179.307,5.959,148.860
C08865=1183.421,60.828,-48.444,-179.310,5.958,148.860
C08866=1183.426,60.578,-48.428,-179.313,5.957,148.861
C08867=1183.430,60.329,-48.411,-179.315,5.956,148.861
C08868=1183.436,60.080,-48.395,-179.318,5.955,148.862
C08869=1183.440,59.831,-48.378,-179.320,5.954,148.862
C08870=1183.446,59.580,-48.362,-179.323,5.953,148.863
C08871=1183.451,59.331,-48.345,-179.326,5.953,148.864
C08872=1183.455,59.082,-48.329,-179.328,5.951,148.864
C08873=1183.461,58.833,-48.313,-179.331,5.950,148.865
C08874=1183.465,58.583,-48.297,-179.333,5.949,148.865
C08875=1183.470,58.334,-48.280,-179.336,5.949,148.866
C08876=1183.476,58.084,-48.264,-179.338,5.947,148.866
C08877=1183.481,57.835,-48.247,-179.341,5.947,148.867
C08878=1183.485,57.586,-48.231,-179.344,5.946,148.867
C08879=1183.491,57.336,-48.215,-179.346,5.945,148.868
C08880=1183.495,57.087,-48.198,-179.349,5.944,148.869
C08881=1183.500,56.837,-48.183,-179.351,5.943,148.869
C08882=1183.505,56.588,-48.166,-179.354,5.943,148.870
C08883=1183.510,56.339,-48.150,-179.357,5.941,148.870
C08884=1183.515,56.089,-48.134,-179.359,5.940,148.871
C08885=1183.520,55.840,-48.118,-179.362,5.940,148.871
C08886=1183.525,55.590,-48.101,-179.364,5.939,148.872
C08887=1183.530,55.341,-48.085,-179.367,5.938,148.873
C08888=1183.535,55.091,-48.069,-179.370,5.937,148.873
C08889=1183.540,54.823,-48.051,-179.372,5.936,148.874
C08890=1183.545,54.554,-48.034,-179.375,5.935,148.874
C08891=1183.551,54.285,-48.017,-179.378,5.934,148.875
C08892=1183.556,54.017,-47.999,-179.381,5.933,148.876
C08893=1183.561,53.767,-47.983,-179.383,5.932,148.876
C08894=1183.566,53.519,-47.967,-179.386,5.932,148.877
C08895=1183.571,53.268,-47.951,-179.388,5.931,148.877
C08896=1183.576,53.020,-47.934,-179.391,5.929,148.878
C08897=1183.581,52.770,-47.919,-179.394,5.929,148.879
C08898=1183.586,52.520,-47.903,-179.396,5.928,148.879
C08899=1183.591,52.271,-47.887,-179.399,5.928,148.880
C08900=1183.596,52.021,-47.871,-179.402,5.926,148.880
C08901=1183.601,51.773,-47.854,-179.404,5.925,148.881
C08902=1183.606,51.522,-47.838,-179.407,5.925,148.881
C08903=1183.611,51.274,-47.822,-179.409,5.924,148.882
C08904=1183.616,51.024,-47.806,-179.412,5.923,148.883
C08905=1183.621,50.774,-47.791,-179.415,5.922,148.883
C08906=1183.626,50.525,-47.774,-179.417,5.921,148.884
C08907=1183.631,50.275,-47.758,-179.419,5.921,148.884
C08908=1183.636,50.026,-47.742,-179.422,5.919,148.885
C08909=1183.640,49.777,-47.727,-179.425,5.918,148.885
C08910=1183.646,49.527,-47.711,-179.427,5.918,148.886
C08911=1183.651,49.278,-47.695,-179.430,5.917,148.887
C08912=1183.655,49.028,-47.679,-179.432,5.917,148.887
C08913=1183.661,48.779,-47.663,-179.435,5.915,148.888
C08914=1183.666,48.529,-47.647,-179.438,5.914,148.888
C08915=1183.671,48.280,-47.631,-179.440,5.914,148.889
C08916=1183.676,48.031,-47.615,-179.442,5.913,148.889
C08917=1183.681,47.781,-47.599,-179.446,5.912,148.890
C08918=1183.685,47.532,-47.584,-179.448,5.911,148.891
C08919=1183.691,47.283,-47.568,-179.450,5.910,148.891
C08920=1183.695,47.033,-47.552,-179.453,5.910,148.892
C08921=1183.701,46.783,-47.537,-179.456,5.909,148.893
C08922=1183.705,46.534,-47.520,-179.458,5.908,148.893
C08923=1183.711,46.284,-47.504,-179.461,5.907,148.894
C08924=1183.715,46.035,-47.489,-179.463,5.906,148.894
C08925=1183.720,45.785,-47.473,-179.466,5.906,148.895
C08926=1183.725,45.536,-47.457,-179.469,5.904,148.895
C08927=1183.731,45.287,-47.441,-179.471,5.903,148.896
C08928=1183.735,45.037,-47.426,-179.474,5.903,148.897
C08929=1183.740,44.788,-47.411,-179.477,5.902,148.897
C08930=1183.745,44.538,-47.395,-179.479,5.902,148.898
C08931=1183.751,44.289,-47.379,-179.482,5.900,148.898
C08932=1183.755,44.039,-47.363,-179.484,5.899,148.899
C08933=1183.761,43.790,-47.347,-179.487,5.899,148.899
C08934=1183.765,43.541,-47.332,-179.489,5.898,148.900
C08935=1183.770,43.291,-47.316,-179.492,5.897,148.901
C08936=1183.775,43.041,-47.301,-179.495,5.896,148.901
C08937=1183.781,42.792,-47.285,-179.497,5.896,148.902
C08938=1183.785,42.542,-47.270,-179.500,5.895,148.902
C08939=1183.790,42.293,-47.254,-179.502,5.894,148.903
C08940=1183.796,42.043,-47.238,-179.504,5.893,148.903
C08941=1183.801,41.794,-47.223,-179.507,5.893,148.904
C08942=1183.805,41.545,-47.207,-179.510,5.892,148.905
C08943=1183.810,41.295,-47.191,-179.512,5.891,148.905
C08944=1183.816,41.046,-47.176,-179.515,5.890,148.906
C08945=1183.820,40.797,-47.161,-179.518,5.890,148.907
C08946=1183.825,40.547,-47.145,-179.520,5.889,148.907
C08947=1183.830,40.297,-47.129,-179.523,5.887,148.908
C08948=1183.835,40.048,-47.114,-179.526,5.887,148.908
C08949=1183.840,39.799,-47.098,-179.528,5.886,148.909
C08950=1183.845,39.549,-47.083,-179.530,5.886,148.909
C08951=1183.850,39.300,-47.068,-179.533,5.885,148.910
C08952=1183.855,39.050,-47.052,-179.535,5.884,148.911
C08953=1183.861,38.801,-47.036,-179.538,5.883,148.911
C08954=1183.865,38.551,-47.021,-179.541,5.882,148.912
C08955=1183.870,38.301,-47.006,-179.543,5.881,148.912
C08956=1183.876,38.052,-46.991,-179.546,5.881,148.913
C08957=1183.880,37.803,-46.976,-179.548,5.880,148.914
C08958=1183.886,37.553,-46.960,-179.551,5.880,148.914
C08959=1183.891,37.303,-46.944,-179.554,5.878,148.915
C08960=1183.895,37.054,-46.929,-179.556,5.877,148.915
C08961=1183.901,36.805,-46.913,-179.559,5.877,148.916
C08962=1183.905,36.556,-46.898,-179.561,5.876,148.917
C08963=1183.911,36.306,-46.883,-179.564,5.876,148.917
C08964=1183.916,36.057,-46.867,-179.566,5.875,148.918
C08965=1183.920,35.806,-46.853,-179.569,5.874,148.918
C08966=1183.926,35.557,-46.837,-179.572,5.873,148.919
C08967=1183.930,35.308,-46.822,-179.574,5.872,148.920
C08968=1183.936,35.058,-46.806,-179.577,5.872,148.920
C08969=1183.940,34.809,-46.791,-179.579,5.871,148.921
C08970=1183.946,34.560,-46.776,-179.582,5.870,148.921
C08971=1183.950,34.310,-46.761,-179.584,5.870,148.922
C08972=1183.956,34.060,-46.746,-179.587,5.868,148.922
C08973=1183.960,33.811,-46.731,-179.590,5.868,148.923
C08974=1183.966,33.562,-46.715,-179.592,5.867,148.924
C08975=1183.971,33.312,-46.700,-179.594,5.866,148.924
C08976=1183.976,33.063,-46.685,-179.597,5.866,148.925
C08977=1183.981,32.813,-46.670,-179.600,5.865,148.926
C08978=1183.985,32.563,-46.654,-179.602,5.865,148.926
C08979=1183.990,32.314,-46.640,-179.605,5.864,148.927
C08980=1183.996,32.064,-46.624,-179.608,5.863,148.927
C08981=1184.000,31.815,-46.609,-179.610,5.862,148.928
C08982=1184.006,31.566,-46.594,-179.613,5.861,148.929
C08983=1184.011,31.316,-46.580,-179.615,5.861,148.929
C08984=1184.016,31.067,-46.564,-179.617,5.860,148.930
C08985=1184.021,30.818,-46.549,-179.620,5.860,148.930
C08986=1184.026,30.568,-46.534,-179.623,5.859,148.931
C08987=1184.031,30.318,-46.519,-179.625,5.858,148.932
C08988=1184.036,30.068,-46.503,-179.628,5.857,148.932
C08989=1184.041,29.819,-46.489,-179.631,5.856,148.933
C08990=1184.045,29.570,-46.474,-179.633,5.855,148.933
C08991=1184.051,29.320,-46.458,-179.636,5.855,148.934
C08992=1184.056,29.070,-46.444,-179.638,5.854,148.935
C08993=1184.062,28.801,-46.428,-179.640,5.854,148.935
C08994=1184.066,28.533,-46.411,-179.644,5.852,148.936
C08995=1184.072,28.264,-46.395,-179.646,5.852,148.936
C08996=1184.077,27.995,-46.379,-179.649,5.851,148.937
C08997=1184.082,27.746,-46.364,-179.651,5.851,148.938
C08998=1184.088,27.496,-46.349,-179.654,5.850,148.938
C08999=1184.092,27.247,-46.334,-179.656,5.849,148.939
C09000=1184.098,26.997,-46.320,-179.660,5.848,148.940
C09001=1184.103,26.748,-46.305,-179.662,5.847,148.940
C09002=1184.108,26.498,-46.290,-179.664,5.847,148.941
C09003=1184.113,26.249,-46.275,-179.667,5.846,148.941
C09004=1184.118,25.999,-46.260,-179.669,5.845,148.942
C09005=1184.123,25.750,-46.245,-179.672,5.845,148.943
C09006=1184.128,25.500,-46.231,-179.674,5.844,148.943
C09007=1184.133,25.251,-46.216,-179.677,5.844,148.944
C09008=1184.138,25.001,-46.201,-179.679,5.843,148.944
C09009=1184.143,24.752,-46.186,-179.682,5.843,148.945
C09010=1184.148,24.502,-46.171,-179.685,5.841,148.946
C09011=1184.153,24.253,-46.156,-179.687,5.840,148.946
C09012=1184.158,24.003,-46.142,-179.690,5.840,148.947
C09013=1184.163,23.754,-46.127,-179.693,5.839,148.948
C09014=1184.168,23.504,-46.112,-179.695,5.839,148.948
C09015=1184.173,23.254,-46.098,-179.697,5.838,148.949
C09016=1184.178,23.005,-46.083,-179.700,5.838,148.949
C09017=1184.184,22.755,-46.068,-179.702,5.837,148.950
C09018=1184.188,22.506,-46.053,-179.705,5.836,148.950
C09019=1184.193,22.257,-46.039,-179.707,5.836,148.951
C09020=1184.198,22.007,-46.025,-179.710,5.835,148.952
C09021=1184.204,21.757,-46.009,-179.712,5.834,148.952
C09022=1184.209,21.508,-45.995,-179.716,5.833,148.953
C09023=1184.213,21.258,-45.980,-179.718,5.832,148.953
C09024=1184.218,21.009,-45.965,-179.720,5.832,148.954
C09025=1184.224,20.759,-45.951,-179.723,5.831,148.955
C09026=1184.229,20.511,-45.936,-179.725,5.830,148.955
C09027=1184.234,20.261,-45.922,-179.728,5.830,148.956
C09028=1184.239,20.011,-45.907,-179.730,5.829,148.957
C09029=1184.244,19.761,-45.893,-179.733,5.829,148.957
C09030=1184.249,19.512,-45.878,-179.735,5.828,148.958
C09031=1184.254,19.262,-45.863,-179.738,5.828,148.958
C09032=1184.259,19.013,-45.849,-179.741,5.827,148.959
C09033=1184.264,18.763,-45.834,-179.743,5.826,148.960
C09034=1184.269,18.514,-45.820,-179.745,5.826,148.960
C09035=1184.274,18.264,-45.805,-179.748,5.825,148.961
C09036=1184.279,18.014,-45.791,-179.750,5.824,148.961
C09037=1184.285,17.766,-45.776,-179.753,5.824,148.962
C09038=1184.290,17.516,-45.762,-179.755,5.823,148.963
C09039=1184.295,17.266,-45.747,-179.758,5.822,148.963
C09040=1184.300,17.017,-45.733,-179.761,5.821,148.964
C09041=1184.305,16.767,-45.719,-179.764,5.821,148.965
C09042=1184.309,16.518,-45.704,-179.766,5.820,148.965
C09043=1184.314,16.268,-45.690,-179.768,5.819,148.966
C09044=1184.319,16.018,-45.675,-179.771,5.819,148.966
C09045=1184.325,15.769,-45.661,-179.774,5.818,148.967
C09046=1184.330,15.520,-45.647,-179.776,5.818,148.968
C09047=1184.335,15.270,-45.632,-179.778,5.817,148.968
C09048=1184.340,15.020,-45.617,-179.781,5.817,148.969
C09049=1184.345,14.771,-45.603,-179.783,5.816,148.969
C09050=1184.350,14.521,-45.589,-179.786,5.815,148.970
C09051=1184.355,14.272,-45.575,-179.789,5.815,148.971
C09052=1184.360,14.022,-45.560,-179.791,5.814,148.971
C09053=1184.365,13.773,-45.546,-179.793,5.813,148.972
C09054=1184.370,13.523,-45.532,-179.796,5.813,148.973
C09055=1184.375,13.273,-45.518,-179.799,5.812,148.973
C09056=1184.380,13.023,-45.503,-179.801,5.812,148.974
C09057=1184.386,12.774,-45.489,-179.803,5.811,148.974
C09058=1184.391,12.525,-45.475,-179.806,5.811,148.975
C09059=1184.395,12.276,-45.460,-179.808,5.810,148.976
C09060=1184.400,12.026,-45.446,-179.811,5.809,148.976
C09061=1184.405,11.776,-45.432,-179.814,5.809,148.977
C09062=1184.411,11.527,-45.418,-179.816,5.808,148.978
C09063=1184.416,11.278,-45.403,-179.818,5.807,148.978
C09064=1184.421,11.028,-45.389,-179.821,5.807,148.979
C09065=1184.426,10.778,-45.375,-179.824,5.806,148.979
C09066=1184.431,10.529,-45.361,-179.826,5.806,148.980
C09067=1184.436,10.279,-45.347,-179.829,5.805,148.981
C09068=1184.441,10.030,-45.332,-179.831,5.805,148.981
C09069=1184.446,9.780,-45.318,-179.834,5.804,148.982
C09070=1184.452,9.531,-45.304,-179.836,5.803,148.982
C09071=1184.457,9.281,-45.291,-179.839,5.803,148.983
C09072=1184.462,9.031,-45.276,-179.841,5.802,148.984
C09073=1184.466,8.782,-45.263,-179.843,5.801,148.984
C09074=1184.472,8.532,-45.249,-179.846,5.801,148.985
C09075=1184.477,8.283,-45.234,-179.849,5.801,148.986
C09076=1184.482,8.033,-45.220,-179.851,5.800,148.986
C09077=1184.487,7.783,-45.206,-179.854,5.799,148.987
C09078=1184.492,7.534,-45.192,-179.856,5.799,148.987
C09079=1184.497,7.285,-45.178,-179.859,5.798,148.988
C09080=1184.502,7.035,-45.163,-179.861,5.797,148.989
C09081=1184.507,6.785,-45.149,-179.864,5.797,148.989
C09082=1184.513,6.536,-45.136,-179.866,5.796,148.990
C09083=1184.517,6.286,-45.122,-179.869,5.796,148.990
C09084=1184.522,6.036,-45.108,-179.871,5.795,148.991
C09085=1184.528,5.787,-45.094,-179.874,5.795,148.992
C09086=1184.532,5.538,-45.080,-179.876,5.794,148.992
C09087=1184.537,5.288,-45.066,-179.879,5.793,148.993
C09088=1184.543,5.038,-45.052,-179.881,5.793,148.994
C09089=1184.548,4.789,-45.039,-179.884,5.792,148.994
C09090=1184.552,4.539,-45.024,-179.886,5.791,148.995
C09091=1184.557,4.290,-45.010,-179.889,5.791,148.995
C09092=1184.563,4.040,-44.997,-179.891,5.791,148.996
C09093=1184.568,3.790,-44.983,-179.894,5.790,148.997
C09094=1184.572,3.541,-44.969,-179.896,5.789,148.997
C09095=1184.578,3.292,-44.955,-179.899,5.789,148.998
C09096=1184.583,3.042,-44.941,-179.902,5.788,148.999
C09097=1184.588,2.773,-44.926,-179.904,5.788,148.999
C09098=1184.594,2.504,-44.911,-179.907,5.787,149.000
C09099=1184.600,2.235,-44.896,-179.910,5.786,149.001
C09100=1184.605,1.965,-44.881,-179.912,5.785,149.001
C09101=1184.610,1.715,-44.868,-179.915,5.785,149.002
C09102=1184.615,1.466,-44.854,-179.918,5.784,149.003
C09103=1184.620,1.216,-44.840,-179.920,5.784,149.003
C09104=1184.626,0.966,-44.826,-179.922,5.783,149.004
C09105=1184.630,0.717,-44.813,-179.925,5.782,149.004
C09106=1184.635,0.468,-44.799,-179.928,5.782,149.005
C09107=1184.641,0.218,-44.786,-179.930,5.781,149.006
C09108=1184.646,-0.032,-44.771,-179.932,5.781,149.006
C09109=1184.650,-0.281,-44.758,-179.935,5.781,149.007
C09110=1184.656,-0.531,-44.745,-179.937,5.780,149.008
C09111=1184.661,-0.780,-44.730,-179.939,5.780,149.008
C09112=1184.666,-1.029,-44.717,-179.942,5.779,149.009
C09113=1184.671,-1.279,-44.703,-179.945,5.779,149.009
C09114=1184.676,-1.529,-44.689,-179.947,5.778,149.010
C09115=1184.682,-1.779,-44.676,-179.950,5.777,149.011
C09116=1184.686,-2.028,-44.662,-179.952,5.777,149.011
C09117=1184.692,-2.278,-44.649,-179.955,5.776,149.012
C09118=1184.697,-2.527,-44.635,-179.957,5.776,149.012
C09119=1184.702,-2.776,-44.621,-179.960,5.775,149.013
C09120=1184.707,-3.027,-44.608,-179.962,5.775,149.014
C09121=1184.711,-3.276,-44.594,-179.965,5.774,149.014
C09122=1184.717,-3.526,-44.581,-179.967,5.773,149.015
C09123=1184.722,-3.775,-44.567,-179.970,5.773,149.016
C09124=1184.727,-4.025,-44.554,-179.972,5.772,149.016
C09125=1184.732,-4.274,-44.540,-179.975,5.771,149.017
C09126=1184.738,-4.524,-44.527,-179.977,5.771,149.017
C09127=1184.742,-4.773,-44.513,-179.979,5.771,149.018
C09128=1184.748,-5.023,-44.500,-179.982,5.771,149.019
C09129=1184.753,-5.272,-44.486,-179.984,5.770,149.019
C09130=1184.758,-5.522,-44.473,-179.987,5.770,149.020
C09131=1184.763,-5.772,-44.459,-179.990,5.769,149.021
C09132=1184.768,-6.021,-44.446,-179.992,5.769,149.021
C09133=1184.774,-6.271,-44.432,-179.994,5.768,149.022
C09134=1184.779,-6.520,-44.419,-179.997,5.767,149.023
C09135=1184.784,-6.770,-44.406,-180.000,5.767,149.023
C09136=1184.789,-7.019,-44.392,179.998,5.766,149.024
C09137=1184.794,-7.269,-44.379,179.996,5.766,149.024
C09138=1184.799,-7.518,-44.365,179.993,5.765,149.025
C09139=1184.804,-7.768,-44.352,179.990,5.765,149.026
C09140=1184.810,-8.018,-44.339,179.988,5.764,149.026
C09141=1184.814,-8.267,-44.325,179.986,5.764,149.027
C09142=1184.820,-8.517,-44.312,179.983,5.764,149.028
C09143=1184.824,-8.767,-44.299,179.981,5.763,149.028
C09144=1184.830,-9.016,-44.285,179.978,5.762,149.029
C09145=1184.834,-9.266,-44.272,179.976,5.762,149.029
C09146=1184.840,-9.516,-44.259,179.973,5.761,149.030
C09147=1184.845,-9.765,-44.245,179.971,5.761,149.031
C09148=1184.850,-10.015,-44.232,179.968,5.760,149.031
C09149=1184.855,-10.265,-44.219,179.966,5.760,149.032
C09150=1184.860,-10.514,-44.205,179.963,5.759,149.033
